nIndex := 0;
IF ipListOfMoversToCheck <> 0 THEN
	THIS^.ipListOfMoversToCheck.ResetIterator();
	WHILE THIS^.ipListOfMoversToCheck.HasNextObject() DO
		
		//Cheack all Movers fill the actposition in the array
		IF ToXpMover(THIS^.ipListOfMoversToCheck.GetNextObject(),ipMover) THEN
			aMoversInterfaceLastCycle[nIndex] 	:= ipMover;
			aMoversPositionLastCycle[nIndex] 	:= ipMover.PositionOnTrack;
			aMoversTrackLastCycle[nIndex]		:= ipMover.CurrentTrack;
			nIndex := nIndex +1;
		END_IF
		
	END_WHILE	
	THIS^.ipListOfMoversToCheck.RestoreIterator();
END_IF
END_METHOD

END_FUNCTION_BLOCK

// COMPONENTs/Optional/Trigger/I_XP_Trigger
INTERFACE I_XP_Trigger  EXTENDS __SYSTEM.IQueryInterface

{attribute 'monitoring':='call'}
PROPERTY AccocietedTrack : I_XP_Track
GET
END_GET
SET
END_SET
END_PROPERTY

{attribute 'monitoring':='call'}
PROPERTY HR : HRESULT
GET
END_GET
END_PROPERTY

PROPERTY ListOfMoversToCheck : I_CH_List
SET
END_SET
END_PROPERTY

{attribute 'monitoring':='call'}
PROPERTY MoverAtTrigger : I_XP_Mover
GET
END_GET
END_PROPERTY

{attribute 'monitoring':='call'}
PROPERTY MoverDetected : BOOL
GET
END_GET
END_PROPERTY

{attribute 'monitoring':='call'}
PROPERTY PositionOnTrack : LREAL
GET
END_GET
SET
END_SET
END_PROPERTY

{attribute 'monitoring':='call'}
PROPERTY TimeStamp : T_DCTIME64;
GET
END_GET
END_PROPERTY

{attribute 'monitoring':='call'}
PROPERTY TriggerDirection : Tc3_Mc3Definitions.MC_Direction
GET
END_GET
SET
END_SET
END_PROPERTY

END_INTERFACE

// COMPONENTs/Optional/Zone/FB_XP_SoretedListOfMover
{attribute 'no_explicit_call' := 'Do not call the body - Stick to OOP'}
// Check zone start to end in positive direktion.
FUNCTION_BLOCK FB_XP_SoretedListOfMover EXTENDS FB_CH_Object IMPLEMENTS I_XP_Zone
VAR
	{attribute 'hide'}
	bInitDone : BOOL;
	{attribute 'hide'}
	ipXpStation : I_XP_Station; //Interface to XPlanar station 
	{attribute 'hide'}
	ipListOfMoversToCheck : CHALET_BaseComponents.I_CH_LIST;
	{attribute 'hide'}
	aMoversInZone : ARRAY [0..(CHALET_BaseComponents.BaseParameterlist.MAX_OBJECTS-1)] OF I_XP_Mover_PLC;
END_VAR

{attribute 'monitoring':='call'}
PROPERTY CtsMoversInZone : UINT
GET
VAR
	nIndex : UDINT;
END_VAR
THIS^.Prepare();//Prepare Time-critical information

//Check array for entrys, exit if fisrt empty arrayindex is found.
FOR nIndex := 0 TO (CHALET_BaseComponents.BaseParameterlist.MAX_OBJECTS-1) DO
	IF (aMoversInZone[nIndex] <> 0) THEN
		CtsMoversInZone := CtsMoversInZone +1;
	ELSE
		RETURN;
	END_IF
END_FOR
END_GET
END_PROPERTY

METHOD FB_init : BOOL
VAR_INPUT
	bInitRetains : BOOL; // if TRUE, the retain variables are initialized (warm start / cold start)
	bInCopyCode : BOOL;  // if TRUE, the instance afterwards gets moved into the copy code (online change)
	
	ipXpStation : I_XP_Station; //Interface to XPlanar station 
	ipListOfMoversToCheck : CHALET_BaseComponents.I_CH_LIST;
END_VAR
VAR_INST
	{attribute 'hide'}
	bFBInitCalledOnce : BOOL; //Do the following code once during start up and not during onlinechange
END_VAR
//Do the following code once during start up and not during onlinechange
IF NOT bFBInitCalledOnce THEN 
	;
END_IF

THIS^.ipXpStation := ipXpStation;
THIS^.ipListOfMoversToCheck := ipListOfMoversToCheck;


bFBInitCalledOnce := TRUE;
END_METHOD

METHOD Initialize : HRESULT
IF THIS^.ipXpStation = 0 THEN
	//No valide interface
	Initialize := E_FAIL;
	RETURN;
END_IF

IF THIS^.ipListOfMoversToCheck = 0 THEN
	//No valide interface
	Initialize := E_FAIL;
	RETURN;
END_IF


bInitDone := TRUE;
Initialize := S_OK;
END_METHOD

{attribute 'monitoring':='call'}
// Return a sorted list of movers in this zone. Index 0 is the mover in Front.
PROPERTY MoversInZone : REFERENCE TO ARRAY [0..(CHALET_BaseComponents.BaseParameterlist.MAX_OBJECTS-1)] OF I_XP_Mover_PLC
GET
THIS^.Prepare();//Prepare Time-critical information

MoversInZone REF= THIS^.aMoversInZone;
END_GET
END_PROPERTY

(* Time-critical information is processed here, which can then be polled via the property every cycle. 
The update method is usually at the end of the program and then it is already 'outdated'. *)
METHOD PRIVATE Prepare : HRESULT
VAR
	nLoopIndex : UDINT;
	ipMoverPlc : I_XP_Mover_PLC;
	ipMover : I_XP_Mover;
	ipPath : I_XP_Path;
	fDistToStart : LREAL;
	aDisanceToStart : ARRAY [0..(CHALET_BaseComponents.BaseParameterlist.MAX_OBJECTS-1)] OF LREAL;
END_VAR
VAR_INST
	{attribute 'hide'}
	nLastUpdatedCycleCount : UDINT;
END_VAR
IF NOT bInitDone OR ipXpStation.AccocietedTrack = 0 THEN
	Prepare := E_FAIL;
	RETURN;
END_IF

//Check if this Cycle the dates are allready prepared
IF nLastUpdatedCycleCount <> TwinCAT_SystemInfoVarList._TaskInfo[THIS^.nTaskIndex].CycleCount THEN
	nLastUpdatedCycleCount := TwinCAT_SystemInfoVarList._TaskInfo[THIS^.nTaskIndex].CycleCount;

	//Clear array
	MEMSET(destAddr:=ADR(aMoversInZone),n:=SIZEOF(aMoversInZone),fillByte:=0);
	
	//Cheack all Movers and generate a sorted list of all mover in this zone.
	THIS^.ipListOfMoversToCheck.ResetIterator();
	WHILE THIS^.ipListOfMoversToCheck.HasNextObject() DO
		//Check each mover in this stations list
		IF __QUERYINTERFACE(THIS^.ipListOfMoversToCheck.GetNextObject(),ipMoverPlc) THEN
			
			//mover and distance are known from this point and are now sorted into the array
			fDistToStart := ipMoverPlc.DistToParentStation;
			ipMoverPlc := ipMoverPlc;
			
			//Check array of movers and decide if the current one is closer to 
			FOR nLoopIndex := 0 TO (CHALET_BaseComponents.BaseParameterlist.MAX_OBJECTS-1) DO
				//empty array position
				IF aMoversInZone[nLoopIndex] = 0 THEN
					aMoversInZone[nLoopIndex] := ipMoverPlc;
					aDisanceToStart[nLoopIndex] := fDistToStart;
					EXIT;
					
				//Closer Mover found, move whole array 	
				ELSIF aDisanceToStart[nLoopIndex] > fDistToStart THEN
					MEMMOVE(srcAddr := ADR(aMoversInZone[nLoopIndex]), destAddr := ADR(aMoversInZone[nLoopIndex+1]), n := (SIZEOF(aMoversInZone[0])*(CHALET_BaseComponents.BaseParameterlist.MAX_OBJECTS-1-nLoopIndex)));
					MEMMOVE(srcAddr := ADR(aDisanceToStart[nLoopIndex]), destAddr := ADR(aDisanceToStart[nLoopIndex+1]), n := (SIZEOF(aDisanceToStart[0])*(CHALET_BaseComponents.BaseParameterlist.MAX_OBJECTS-1-nLoopIndex)));
					aMoversInZone[nLoopIndex] := ipMoverPlc;
					aDisanceToStart[nLoopIndex] := fDistToStart;
					EXIT;
					
				//check next position	
				ELSE 
					;
				END_IF
			END_FOR
		END_IF
	END_WHILE
	THIS^.ipListOfMoversToCheck.RestoreIterator();
END_IF
END_METHOD

METHOD Update : HRESULT
VAR

END_VAR
// Nothing todo in Update. Check Prepare
END_METHOD

END_FUNCTION_BLOCK

// COMPONENTs/Optional/Zone/I_XP_Zone
INTERFACE I_XP_Zone

{attribute 'monitoring':='call'}
PROPERTY CtsMoversInZone : UINT
GET
END_GET
END_PROPERTY

{attribute 'monitoring':='call'}
PROPERTY MoversInZone : REFERENCE TO ARRAY [0..(CHALET_BaseComponents.BaseParameterlist.MAX_OBJECTS-1)] OF I_XP_Mover_PLC // Return a sorted list of movers in this zone. Index 0 is the mover in Front.
GET
END_GET
END_PROPERTY

END_INTERFACE

// COMPONENTs/Optional/I_XP_Path
INTERFACE I_XP_Path  EXTENDS __SYSTEM.IQueryInterface, I_CH_Object

METHOD DistanceToDestiantion : LREAL
VAR_INPUT
	ipTrack : I_XP_Track;
	fPosOnTrack : LREAL;
END_VAR
END_METHOD

{attribute 'monitoring':='call'}
PROPERTY Length : LREAL
GET
END_GET
SET
END_SET
END_PROPERTY

PROPERTY PointerToThis : POINTER TO FB_XP_Path
GET
END_GET
END_PROPERTY

{attribute 'monitoring':='call'}
PROPERTY StationDestination : I_XP_Station
GET
END_GET
SET
END_SET
END_PROPERTY

{attribute 'monitoring':='call'}
PROPERTY StationStart  : I_XP_Station
GET
END_GET
SET
END_SET
END_PROPERTY

{attribute 'monitoring':='call'}
PROPERTY TracksUsed : REFERENCE TO FB_CH_List
GET
END_GET
END_PROPERTY

END_INTERFACE

// COMPONENTs/Optional/FB_XP_Path
{attribute 'enable_dynamic_creation'}
{attribute 'no_explicit_call' := 'Do not call the body - Stick to OOP'}
FUNCTION_BLOCK FB_XP_Path EXTENDS FB_CH_Object IMPLEMENTS I_XP_Path
VAR
	fbTracksUsed : FB_CH_List;
	ipStartStation, ipDestinationStation : I_XP_Station;
	fPathLength : LREAL;
END_VAR

METHOD DistanceToDestiantion : LREAL
VAR_INPUT
	ipTrack : I_XP_Track;
	fPosOnTrack : LREAL;
END_VAR
VAR
	ipTrackTemp : I_XP_Track; 
	bStartTrackFound : BOOL := FALSE;
END_VAR
IF ipTrack = 0 THEN
	//Error -  invalide interface
	DistanceToDestiantion := CHALET_BaseComponents.GVL_Datatypes.cMaxLreal;
	RETURN;
END_IF

IF NOT fbTracksUsed.FindObject(ipTrack) OR fPosOnTrack < 0 OR  fPosOnTrack > ipTrack.Length THEN
	//Error -  position not on track
	DistanceToDestiantion := CHALET_BaseComponents.GVL_Datatypes.cMaxLreal;
	RETURN;
END_IF

//the whole thing works because the tracklist is sorted from start to finish
fbTracksUsed.ResetIterator();
WHILE fbTracksUsed.HasNextObject() DO
	IF ToXpTrack(fbTracksUsed.GetNextObject(),ipTrackTemp) THEN
		//start countion on requestet track
		IF ipTrackTemp = ipTrack OR bStartTrackFound THEN
			bStartTrackFound := TRUE;
			DistanceToDestiantion := DistanceToDestiantion + ipTrackTemp.Length;
 		END_IF
	END_IF
END_WHILE	

DistanceToDestiantion := DistanceToDestiantion - fPosOnTrack;
DistanceToDestiantion := DistanceToDestiantion - THIS^.StationDestination.AccocietedTrack.Length + THIS^.StationDestination.PositionOnTrack;
END_METHOD

{attribute 'monitoring':='call'}
PROPERTY Length : LREAL
GET
Length := THIS^.fPathLength;
END_GET
SET
THIS^.fPathLength := Length;
END_SET
END_PROPERTY

{attribute 'monitoring':='call'}
PROPERTY LUID : STRING //Locally unique identifier
GET
VAR
	sTempName : STRING;
END_VAR
IF ipStartStation <> 0 AND ipDestinationStation <> 0 THEN
	sTempName := CONCAT(sTempName, ipStartStation.LUID);
	sTempName := CONCAT(sTempName, ' to ' );
	sTempName := CONCAT(sTempName, ipDestinationStation.LUID);
	
ELSIF ipStartStation <> 0 THEN
	sTempName := CONCAT(sTempName, ipStartStation.LUID);
	sTempName := CONCAT(sTempName, ' to ?' );

ELSIF ipDestinationStation <> 0 THEN
	sTempName := CONCAT(sTempName, '? to ' );
	sTempName := CONCAT(sTempName, ipDestinationStation.LUID);
	
ELSE 
	sTempName := ' Unknown path';
END_IF


LUID := sTempName;
END_GET
END_PROPERTY

PROPERTY PointerToThis : POINTER TO FB_XP_Path
GET
PointerToThis := ADR(THIS^);
END_GET
END_PROPERTY

{attribute 'monitoring':='call'}
PROPERTY StationDestination : I_XP_Station
GET
StationDestination := THIS^.ipDestinationStation;
END_GET
SET
THIS^.ipDestinationStation := StationDestination;
END_SET
END_PROPERTY

{attribute 'monitoring':='call'}
PROPERTY StationStart  : I_XP_Station
GET
StationStart := THIS^.ipStartStation;
END_GET
SET
THIS^.ipStartStation := StationStart;
END_SET
END_PROPERTY

{attribute 'monitoring':='call'}
PROPERTY TracksUsed : REFERENCE TO FB_CH_List
GET
TracksUsed REF= THIS^.fbTracksUsed;
END_GET
END_PROPERTY

END_FUNCTION_BLOCK

// COMPONENTs/Optional/F_GetDistToPosModulo
FUNCTION F_GetDistToPosModulo : LREAL //This is only working in Positiv Direktion
VAR_INPUT
	fTargedPosition : LREAL;
	fActualPosition : LREAL;
	fModulo 		: LREAL;
END_VAR

VAR

END_VAR

IF fTargedPosition < fActualPosition THEN
	fTargedPosition := fTargedPosition + fModulo;
END_IF

F_GetDistToPosModulo := fTargedPosition - fActualPosition;

END_FUNCTION

// COMPONENTs/Optional/F_InLimitTest
FUNCTION F_InLimitTest : BOOL
VAR_INPUT
	fMinimum 	: LREAL;
	fMaximum 	: LREAL;
	fInput 		: LREAL;
END_VAR

//Normal case
// 9 Max
// 5 Test
// 1 Min
IF fMinimum <= fMaximum THEN
	F_InLimitTest := (fInput >= fMinimum) AND (fInput <= fMaximum);
	
//Modulo case	
// 6 | 6  Max
// 5 | 9  Test
// 8 | 8  Min
ELSIF fMinimum > fMaximum THEN
	F_InLimitTest := NOT((fInput > fMaximum) AND (fInput < fMinimum));
END_IF

END_FUNCTION

// COMPONENTs/Stationen/FB_XP_Station
{attribute 'no_explicit_call' := 'Do not call the body - Stick to OOP'}
(* XPlanar station - n per associated XPlanar. Can be instantiated as an array and/or individually
	The stations are the main component of the application. As soon as the system has been started up and all movers are on the track, the movers are only sent from one station to the next.
	Parameters:
		xPos, yPos 			= Absolute position of the station on the xPlanar.
		ipAccocietedTrack 	= The track on which the station is located. If the XY position is not on this track, the next possible track position is assumed on this track.
		sUniqueName 		= Unique name that may only exist once.
		sTargetGroup 		= A name for a group to which this station belongs. Important for redundant stations
 *)	
FUNCTION_BLOCK FB_XP_Station EXTENDS FB_CH_Object IMPLEMENTS I_XP_Station, I_XP_Station_PLC
VAR
	//optional - To visualize the station position in LiveView
	fbOptionalTrackUsedInLiveView : MC_PlanarTrack;

	{attribute 'hide'}
	bErrorDuringFbInit : BOOL;	//Fatal error - Not possible to reset
	
	{attribute 'hide'}
	bInitDone : BOOL;
	{attribute 'hide'}	
	bTrackIsSetInFbInit : BOOL;
	{attribute 'hide'}	
	bMoversInPlace : BOOL;
	{attribute 'hide'}                   	
	eActiveCommand 		: CHALET_Nc.E_NcAxisCommands := CHALET_Nc.E_NcAxisCommands.None;
	{attribute 'hide'}	
	ipXpSystem : I_XP_System_Registration;
	{attribute 'hide'}
	bReadyToRecvMovers 		: BOOL := TRUE;
	{attribute 'hide'}
	sTargetGroup 				: STRING;
	
	{attribute 'hide'}
	bSuppressDynamicsChange		: BOOL; // Suppress to change the dynamic(Gap+velocity) of passing movers. This is usefull in startup
	{attribute 'hide'}
	fMoverGapAtExit 			: LREAL := XPlanarParameterlist.F_MOVER_MINIMUM_GAP_ON_TRACK; // Every mover that leaves or passes the station gets this new gap as a target.
	{attribute 'hide'}
	fMoverVelocityAtExit		: LREAL; // Every mover that leaves or passes the station gets this new velo as a target.
	
	{attribute 'hide'}	
	fbPositionPlanned : PositionXY; //this is the configured/planned position of the station. set via FB_init. If it is not on the track, the PosOnTrackXY is different
	{attribute 'hide'}	
	fPositionOnTrack : LREAL;
	{attribute 'hide'}
	fbPositionOnTrackXY : PositionXY;	
	{attribute 'hide'}	
	nState_Configuring: INT;
	{attribute 'hide'}	
	ipAccocietedTrack : I_XP_Track;
	{attribute 'hide'}
	nMoverQueueSize 			: UINT;
	{attribute 'hide'}
	fTargetPosWindow			: LREAL := 0.05; //[mm]
	{attribute 'hide'}
	tTargetPosMonitoringTime	: TIME := T#0MS;

	
	(*List of stations*)
	{attribute 'hide'}	
	fbStationsAhead : FB_CH_List;
	{attribute 'hide'}	
	fbStationsBehinde : FB_CH_List;
	
	(*List of paths*)
	{attribute 'hide'}	
	fbListPathAhead : FB_CH_List;
	{attribute 'hide'}
	fbListPathBehind : FB_CH_List;
	
	(* Lists to handle the ownership of movers *)
	{attribute 'hide'}
	fbAssignedMovers 			: FB_CH_List;		// Movers approaching the station. This station is the parent of this movers
	{attribute 'hide'}
	fbFeedback : FB_CH_Feedback;	
	
	//Simulation
	{attribute 'hide'}
	fSimulationProcessDuration 	: LREAL; //[s]
	{attribute 'hide'}
	sSimulationTargedStation	: STRING; //GroupID of the targed station to automatic send after the duration
	
	
	//ipXpSystem Is Not Valid at this point, call the konstruktor again in the FB_Init
	{attribute 'hide'}
	fbTrigger 					: FB_XP_Trigger(ipXpSystem);
	{attribute 'hide'}
	fbSortedListMoversInQueue	: FB_XP_SoretedListOfMover(	ipXpStation := THIS^,
															ipListOfMoversToCheck := fbAssignedMovers );
	{attribute 'hide'}
	fDecisionDistance: LREAL;//[mm]
	
	{attribute 'hide'}
	sFilter : STRING;
END_VAR

METHOD PROTECTED CheckInvalideParameter : HRESULT
VAR
 	ipStation : I_XP_Station;
	fbListOfStationsToCheck : FB_CH_List;
END_VAR
//Get a list of all station whitout this station
fbListOfStationsToCheck.Duplicate(THIS^.ipXpSystem.Stations);
fbListOfStationsToCheck.RemoveObject(THIS^);


fbListOfStationsToCheck.ResetIterator();
WHILE fbListOfStationsToCheck.HasNextObject() DO
	IF ToXpStation(fbListOfStationsToCheck.GetNextObject(), ipStation) THEN
		
		//Check for same positions
		IF (ipStation.PositionOnTrack = THIS^.PositionOnTrack) AND (ipStation.AccocietedTrack = THIS^.AccocietedTrack)  THEN
			//Error two stations have same position on track
			CheckInvalideParameter := E_FAIL;
			RETURN;
		END_IF
		
		//Check same unique id
		IF (ipStation.LUID = THIS^.LUID) THEN
			//Error two stations have same unique id
			CheckInvalideParameter := E_FAIL;
			RETURN;
		END_IF
		
		fbListOfStationsToCheck.RemoveObject(ipStation);
	END_IF
END_WHILE
END_METHOD

METHOD protected GetAccocietedTrack : HRESULT
VAR_INPUT
END_VAR

VAR
	ipTrack : I_XP_Track;
	
	fPosOnTrack, fDist	: LREAL;
	fbPositionXYC : PositionXYC;
	fbPositionXY : PositionXY;
	ipClosestTrack : I_XP_Track;
	fDistClosestTrack : LREAL := CHALET_BaseComponents.GVL_Datatypes.cMaxLreal;
END_VAR
//If track is not defind during FB_init, get closest track 
IF NOT bTrackIsSetInFbInit THEN
	THIS^.ipAccocietedTrack := 0;
	THIS^.ipXpSystem.Tracks.ResetIterator();
	WHILE THIS^.ipXpSystem.Tracks.HasNextObject() DO
		IF ToXpTrack(THIS^.ipXpSystem.Tracks.GetNextObject(),ipTrack) THEN 
			
			fPosOnTrack := ipTrack.PlanarTrack.GetArcLengthClosestTo(geometry:= THIS^.fbPositionPlanned);
			//Get the XYC Pos on track
			ipTrack.PlanarTrack.GetPositionAt(fPosOnTrack, fbPositionXYC);
			//Get radius/ distance to positionTarged
			fbPositionXY.x  := THIS^.fbPositionPlanned.x - fbPositionXYC.x;
			fbPositionXY.y  := THIS^.fbPositionPlanned.y - fbPositionXYC.y;
			fDist := fbPositionXY.GetRadius();
			
			IF fDist < fDistClosestTrack THEN
				fDistClosestTrack := fDist;
				ipClosestTrack := ipTrack;
			END_IF
		END_IF
	END_WHILE
	THIS^.ipXpSystem.Tracks.RestoreIterator();
	
	
	THIS^.ipAccocietedTrack := ipClosestTrack;	
END_IF

// Error - No track found
IF THIS^.ipAccocietedTrack = 0 THEN
	GetAccocietedTrack := E_FAIL;
	RETURN;
END_IF
END_METHOD

METHOD GetDecisionDistance : HRESULT
VAR
	fDistToStartOfTrack : LREAL := CHALET_BaseComponents.GVL_Datatypes.cMaxLreal;
	fDistStationBehind : LREAL := CHALET_BaseComponents.GVL_Datatypes.cMaxLreal;
	
	ipPath : I_XP_Path;
END_VAR
(*
As soon as the mover is closer than this distance, the mover can be sent on to the next one if necessary.
This is the distance from the station to the end of the track or the shortest path to this station. Depending on which is closer. This is to ensure that the mover can no longer be overhauled.
*)
fDistToStartOfTrack := THIS^.PositionOnTrack;

THIS^.PathsBehinde.ResetIterator();
WHILE THIS^.PathsBehinde.HasNextObject() DO
	IF __QUERYINTERFACE(THIS^.PathsBehinde.GetNextObject(), ipPath) THEN
		fDistStationBehind := MIN(fDistStationBehind, ipPath.Length);
	END_IF
END_WHILE
THIS^.PathsBehinde.RestoreIterator();

THIS^.fDecisionDistance := CHALET_BaseComponents.GVL_Datatypes.cMaxLreal;
THIS^.fDecisionDistance := MIN(THIS^.fDecisionDistance, fDistToStartOfTrack);
THIS^.fDecisionDistance := MIN(THIS^.fDecisionDistance, fDistStationBehind);

IF THIS^.fDecisionDistance < 1.0 THEN 
	THIS^.fDecisionDistance := 1.0;
END_IF

GetDecisionDistance := S_OK;
END_METHOD

METHOD protected GetPathsAhead : HRESULT
VAR_INPUT
END_VAR

VAR
	fbPathElementsToCheck : FB_CH_List;
	fbListStationsToGetClosest : FB_CH_List;	
	
	
	ipObject 				: I_CH_Object;
	ipStation,ipStation1,ipStation2 	: I_XP_Station;
	ipTrack					: I_XP_Track; 
	ipLastAddedTrack 		: I_XP_Track;
	ipPath 					: I_XP_Path;
	ipPathCurrentLoop  		: I_XP_Path;
	
	
	pFbPath : POINTER TO FB_XP_Path;
	
	fSeachStartPoint : LREAL;
	nIdx : UDINT;
END_VAR
(*
Check whether there is a station further ahead on this track than this one.
If there is no other station on the track, the previous tracks are filled into a list and searched one after the other to see if they have valid stations. 
If the tracks also have no stations, the track before it is added to the list,...
*)

//Clear list, delete dynamic_creation path objects
WHILE NOT fbListPathAhead.IsEmpty DO
	ipObject := fbListPathAhead.GetRandomObject();
	fbListPathAhead.RemoveObject(ipObject);
	
	__QUERYINTERFACE(ipObject, ipPath) ;
	pFbPath := ipPath.PointerToThis;
	__DELETE(pFbPath);
END_WHILE


//new dynamic_creation path objects
pFbPath := __NEW(FB_XP_Path);
//init path
pFbPath^.StationStart := THIS^;
pFbPath^.TracksUsed.ResetIterator();
pFbPath^.TracksUsed.AddObject(THIS^.AccocietedTrack);

//add to list
fbPathElementsToCheck.AddObject(pFbPath^);

//On first pathsearch get an Station who is further ahead than this
fSeachStartPoint := THIS^.PositionOnTrack;



//While list is not empty
WHILE NOT fbPathElementsToCheck.IsEmpty DO
	__QUERYINTERFACE(fbPathElementsToCheck.GetRandomObject(), ipPathCurrentLoop);
	__QUERYINTERFACE(ipPathCurrentLoop.TracksUsed.GetNextObject(),ipLastAddedTrack);
	
	
	//Closed loop
	IF ipLastAddedTrack.ClosedLoop THEN
		//on closed-loop add all stations of this track to list
		fbListStationsToGetClosest.Duplicate(ipLastAddedTrack.StationsOnTrack);
	
		//remove THIS station from list if more than on station is existing
		IF fbListStationsToGetClosest.Size > 1 THEN
			fbListStationsToGetClosest.RemoveObject(THIS^);
		END_IF
	
		
	
	ELSE
		//Not closed loop	
		//Get a List of all stations on track Position > Startpoint
		ipLastAddedTrack.StationsOnTrack.ResetIterator();
		fbListStationsToGetClosest.Clear();
		WHILE ipLastAddedTrack.StationsOnTrack.HasNextObject() DO
			IF ToXpStation(ipLastAddedTrack.StationsOnTrack.GetNextObject(),ipStation) THEN
				//Add all station ahead to list. on closed-loop add all stations of this track to list
				IF ipStation.PositionOnTrack > fSeachStartPoint THEN
					fbListStationsToGetClosest.AddObject(ipStation);
				END_IF
			END_IF
		END_WHILE	
	END_IF
		
	

	
	//Get closest to startpos(0mm)
	WHILE fbListStationsToGetClosest.Size > 1 DO
		fbListStationsToGetClosest.ResetIterator();
		__QUERYINTERFACE(fbListStationsToGetClosest.GetNextObject(),ipStation1);
		__QUERYINTERFACE(fbListStationsToGetClosest.GetNextObject(),ipStation2);
		
		//If station1 is closer to start than station2, remove station2
		IF 		F_GetDistToPosModulo(fTargedPosition := ipStation1.PositionOnTrack, fActualPosition := fSeachStartPoint, fModulo := ipLastAddedTrack.Length) 
			< 	F_GetDistToPosModulo(fTargedPosition := ipStation2.PositionOnTrack, fActualPosition := fSeachStartPoint, fModulo := ipLastAddedTrack.Length) THEN
			fbListStationsToGetClosest.RemoveObject(ipStation2);
		ELSE	
			fbListStationsToGetClosest.RemoveObject(ipStation1);
		END_IF
	END_WHILE
	
	
	IF fbListStationsToGetClosest.Size = 1 THEN
		//Station FOUND
		__QUERYINTERFACE(fbListStationsToGetClosest.GetRandomObject(), ipStation);
		ipPathCurrentLoop.StationDestination := ipStation;
		
		//Calculate Tracklentgh
		ipPathCurrentLoop.TracksUsed.ResetIterator();
		WHILE ipPathCurrentLoop.TracksUsed.HasNextObject() DO
			IF ToXpTrack(ipPathCurrentLoop.TracksUsed.GetNextObject(),ipTrack) THEN
				ipPathCurrentLoop.Length := ipPathCurrentLoop.Length + ipTrack.Length;
			END_IF
		END_WHILE	
		ipPathCurrentLoop.Length := ipPathCurrentLoop.Length - ipPathCurrentLoop.StationStart.PositionOnTrack;
		ipPathCurrentLoop.Length := ipPathCurrentLoop.Length - ipPathCurrentLoop.StationDestination.AccocietedTrack.Length + ipPathCurrentLoop.StationDestination.PositionOnTrack;
		
		fbListPathAhead.AddObject(ipPathCurrentLoop);
		fbPathElementsToCheck.RemoveObject(ipPathCurrentLoop);
	ELSE
		//Station NOT-FOUND, add the subsequent tracks in the list
		ipLastAddedTrack.TracksAhead.ResetIterator();
		WHILE ipLastAddedTrack.TracksAhead.HasNextObject() DO
			ToXpTrack(ipLastAddedTrack.TracksAhead.GetNextObject(), ipTrack);
			//dublicate current path
			pFbPath := __NEW(FB_XP_Path);
			MEMCPY(destAddr := pFbPath, srcAddr := ipPathCurrentLoop.PointerToThis, n := SIZEOF(FB_XP_Path));
			//Add the new track to fresh created path
			pFbPath^.TracksUsed.AddObject(ipTrack);
			//Add to list to check
			fbPathElementsToCheck.AddObject(pFbPath^);
			
		END_WHILE

		
		//delete current path
		fbPathElementsToCheck.RemoveObject(ipPathCurrentLoop);
		pFbPath := ipPathCurrentLoop.PointerToThis;
		__DELETE(pFbPath);
		
	END_IF

	fSeachStartPoint := -0.1;
END_WHILE
END_METHOD

METHOD protected GetPathsBehind : HRESULT
VAR
	ipThisStation : I_XP_Station;
	ipXpStation : I_XP_Station;
	ipPath		: I_XP_Path;
END_VAR
ipThisStation := THIS^;
fbListPathBehind.Clear();

THIS^.fbStationsBehinde.ResetIterator();
WHILE THIS^.fbStationsBehinde.HasNextObject() DO
	IF __QUERYINTERFACE(THIS^.fbStationsBehinde.GetNextObject(),ipXpStation) THEN
		ipXpStation.PathsAhead.ResetIterator();
		WHILE ipXpStation.PathsAhead.HasNextObject() DO
			IF __QUERYINTERFACE(ipXpStation.PathsAhead.GetNextObject(),ipPath) AND_THEN ipPath.StationDestination = ipThisStation THEN
				//add path to this station to list
				fbListPathBehind.AddObject(ipPath);
			END_IF
		END_WHILE	
	END_IF
END_WHILE
END_METHOD

METHOD PROTECTED GetPosOnTrack : HRESULT
VAR
	fbPositionXYC : PositionXYC;
END_VAR
//GetArcLengthClosestTo track
THIS^.fPositionOnTrack := THIS^.ipAccocietedTrack.PlanarTrack.GetArcLengthClosestTo(geometry:= THIS^.fbPositionPlanned);

//Get the XYC Pos on track
THIS^.ipAccocietedTrack.PlanarTrack.GetPositionAt(THIS^.PositionOnTrack, fbPositionXYC);

//XYC -> XY
THIS^.fbPositionOnTrackXY.SetValuesXY(fbPositionXYC.x,fbPositionXYC.y);


//Check for NaN
IF NOT(THIS^.fPositionOnTrack = THIS^.fPositionOnTrack) THEN
	GetPosOnTrack := E_FAIL;
	RETURN;
END_IF
END_METHOD

METHOD PROTECTED GetStationAhead : HRESULT
VAR
	ipPath 		: I_XP_Path;
END_VAR
fbStationsAhead.Clear();


fbListPathAhead.ResetIterator();
WHILE fbListPathAhead.HasNextObject() DO
	IF __QUERYINTERFACE(fbListPathAhead.GetNextObject(),ipPath) THEN
		//add StationDestination to list
		fbStationsAhead.AddObject(ipPath.StationDestination);
	END_IF
END_WHILE
END_METHOD

METHOD PROTECTED GetStationBehinde : HRESULT
VAR_INPUT
END_VAR
VAR
	ipThisStation : I_XP_Station;
	ipXpStation : I_XP_Station;
	ipXpStationAhead : I_XP_Station;
END_VAR
ipThisStation := THIS^;
fbStationsBehinde.Clear();

//Check each Station
THIS^.ipXpSystem.Stations.ResetIterator();
WHILE THIS^.ipXpSystem.Stations.HasNextObject() DO
	IF __QUERYINTERFACE(THIS^.ipXpSystem.Stations.GetNextObject(),ipXpStation) THEN
		//check the list of stations ahead if this station one is existing
		ipXpStation.StationsAhead.ResetIterator();
		WHILE ipXpStation.StationsAhead.HasNextObject() DO
			IF __QUERYINTERFACE(ipXpStation.StationsAhead.GetNextObject(),ipXpStationAhead) AND_THEN (ipXpStationAhead = ipThisStation) THEN
				//add station to list
				fbStationsBehinde.AddObject(ipXpStation);
			END_IF
		END_WHILE	
	END_IF
END_WHILE	
THIS^.ipXpSystem.Stations.RestoreIterator();
END_METHOD

METHOD SetTrackObjName : HRESULT
VAR
	pObject : ITComObject;
	sName : STRING;
END_VAR
FW_ObjMgr_GetObjectInstance(oid:= THIS^.fbOptionalTrackUsedInLiveView.MCTOPLC_STD.TrackOID, iid:= TC_GLOBAL_IID_LIST.IID_ITComObject, pipUnk:= ADR(pObject));
IF pObject <> 0 THEN
	sName := THIS^.LUID;
	pObject.TcSetObjectName(ADR(sName));
END_IF
END_METHOD

//Call this Methode whith seq 0->99, and wait each step until S_OK is returned
METHOD Configure : HRESULT
VAR_INPUT
	nSeq : UINT; //0->100
END_VAR

VAR_INST
	{attribute 'hide'}
	fbFeedback : MC_PlanarFeedback;	
END_VAR
VAR
	bOptionalTrackUsedInLiveViewIsMapped : BOOL;
	fbPositionXYC : PositionXYC;
END_VAR
bOptionalTrackUsedInLiveViewIsMapped := fbOptionalTrackUsedInLiveView.MCTOPLC_STD.TrackOID <> 0;

CASE nSeq OF
	5:	//Get interface of trackobject
		Configure := THIS^.GetAccocietedTrack();	

	10: //Get closest XY-Position on track
		Configure := THIS^.GetPosOnTrack();
		
	11: //Check id is unique and not multiple stations at same position
		Configure := THIS^.CheckInvalideParameter();		
		
		
	13:	//Init Tigger
		fbTrigger.AccocietedTrack := THIS^.AccocietedTrack;
		fbTrigger.PositionOnTrack := THIS^.PositionOnTrack;
		fbTrigger.ListOfMoversToCheck := THIS^.ipXpSystem.Movers;//All mover
		fbTrigger.TriggerDirection := Tc3_Mc3Definitions. MC_DIRECTION.mcDirectionPositive;
		Configure := fbTrigger.Initialize();
	
	14:	//Init Zone		
		Configure := fbSortedListMoversInQueue.Initialize();	
	
	20: //Fill the list of all paths before this station
		Configure := THIS^.GetPathsAhead();		
		
	25: //Fill the list of all stations before this station
		Configure := THIS^.GetStationAhead();

	30: //Fill the list of all paths behinde this station
		Configure := THIS^.GetStationBehinde();	
			
	35: //Fill the list of all stations behinde this station
		Configure := THIS^.GetPathsBehind();

	40: //Determine the distance from which the station can give a new command to a mover
		Configure := THIS^.GetDecisionDistance();
		

//----------------------------------------------------------------		
//The station can optionally be linked to a track object. this track is then displayed in the live view.
//It takes several cycles to prepare the object
	80: IF bOptionalTrackUsedInLiveViewIsMapped THEN
			fbOptionalTrackUsedInLiveView.Clear(fbFeedback);
		END_IF
		
	81:	//Wait for clearing
		IF bOptionalTrackUsedInLiveViewIsMapped THEN
			IF fbFeedback.Done THEN
				Configure := S_OK;
			ELSIF fbFeedback.Busy THEN
				Configure := S_PENDING;
			ELSIF fbFeedback.Error THEN
				Configure := E_FAIL;
			END_IF	
		END_IF

	82: //Set position 
		IF bOptionalTrackUsedInLiveViewIsMapped THEN
			fbPositionXYC.SetValuesXY(THIS^.PositionOnTrackXY.x, THIS^.PositionOnTrackXY.y);
			fbOptionalTrackUsedInLiveView.AppendPosition(position := fbPositionXYC, commandFeedback:= fbFeedback);	
		END_IF	
	
	83:	//Wait for set position
		IF bOptionalTrackUsedInLiveViewIsMapped THEN
			IF fbFeedback.Done THEN
				Configure := S_OK;
			ELSIF fbFeedback.Busy THEN
				Configure := S_PENDING;
			ELSIF fbFeedback.Error THEN
				Configure := E_FAIL;
			END_IF	
		END_IF
		
	84:	//Set name of "track" to stationsname 
		IF bOptionalTrackUsedInLiveViewIsMapped THEN
 			Configure := SetTrackObjName();
		END_IF
//----------------------------------------------------------------

		
		

	100..CHALET_BaseComponents.GVL_Datatypes.cMaxUint: 
		// 100..MaxUint -> Invalide input
		Configure := E_FAIL;
		
	ELSE 
		//If an step is not defind/used return ok
		Configure := S_OK;
END_CASE


fbOptionalTrackUsedInLiveView.Update();
fbFeedback.Update();
END_METHOD

{attribute 'monitoring':='call'}
PROPERTY CtsEmptySpaceInQueue : UDINT
GET
//Handle UINT Overflow
IF THIS^.fbAssignedMovers.Size >= THIS^.nMoverQueueSize THEN
	CtsEmptySpaceInQueue := 0;
ELSE 
	CtsEmptySpaceInQueue := THIS^.nMoverQueueSize - THIS^.fbAssignedMovers.Size;
END_IF
END_GET
END_PROPERTY

{attribute 'monitoring':='call'}
PROPERTY CtsMoversInQueue : UDINT
GET
CtsMoversInQueue := THIS^.fbAssignedMovers.Size;
END_GET
END_PROPERTY

{attribute 'monitoring':='call'}
PROPERTY MoverQueueSize : UINT
GET
MoverQueueSize := THIS^.nMoverQueueSize;
END_GET
SET
THIS^.nMoverQueueSize := MoverQueueSize;
END_SET
END_PROPERTY

{attribute 'monitoring':='call'}
PROPERTY MoversInPlace : BOOL
GET
THIS^.Prepare();//Prepare time-critical information, if not already done


MoversInPlace := bMoversInPlace;
END_GET
END_PROPERTY

{attribute 'monitoring':='call'}
// Return a sorted list of movers in this zone. Index 0 is the mover in Front
PROPERTY MoversInQueue : REFERENCE TO ARRAY [0..(CHALET_BaseComponents.BaseParameterlist.MAX_OBJECTS-1)] OF I_XP_Mover_PLC
GET
MoversInQueue REF= THIS^.fbSortedListMoversInQueue.MoversInZone;
END_GET
END_PROPERTY

{attribute 'monitoring':='call'}
//prevent further movers from entering the station, 
//e.g. to prevent a collision. All movers that are already moving to reach this station will be stopped with a stop 
//and restarted with Ready True.
PROPERTY ReadyToRecvMovers : BOOL
GET
ReadyToRecvMovers := bReadyToRecvMovers;
END_GET
SET
VAR
	ipEachMover : I_XP_Mover;
END_VAR
//Change to Not Ready:
IF (ReadyToRecvMovers = FALSE) AND (bReadyToRecvMovers <> ReadyToRecvMovers) THEN
	//halt all movers on the way
	fbAssignedMovers.ResetIterator();
	WHILE fbAssignedMovers.HasNextObject() DO
		IF ToXpMover(fbAssignedMovers.GetNextObject(),ipEachMover) THEN
			ipEachMover.Halt();	
		END_IF	
	END_WHILE
END_IF

//Change to Ready:
IF (ReadyToRecvMovers = TRUE) AND (bReadyToRecvMovers <> ReadyToRecvMovers) THEN
	//all movers that are on the way have probably been stopped before. when reactivated, the last move command is sent again.
	fbAssignedMovers.ResetIterator();
	WHILE fbAssignedMovers.HasNextObject() DO
		IF ToXpMover(fbAssignedMovers.GetNextObject(),ipEachMover) THEN
			ipEachMover.MoveOnTrack(ipTrack 	:= ipEachMover.LastCmdTargedTrack ,
									fPosition	:= ipEachMover.LastCmdTargedPosition,
									fGap		:= ipEachMover.LastCmdTargedGap);
		END_IF	
	END_WHILE
END_IF

//Store new status
bReadyToRecvMovers := ReadyToRecvMovers;
END_SET
END_PROPERTY

METHOD SendMoversToStation : I_CH_Feedback //All movers in the station are sent to this destination
VAR_INPUT
	sTargetStation: STRING;//unique station name or group of stations
END_VAR
VAR
	nIdx : UDINT;
	ipXpMover : I_XP_Mover;
END_VAR
IF THIS^.fbFeedback.Error THEN
	//Error active/not ready
	THIS^.fbFeedback.LastCommandAccepted	:= FALSE;
	RETURN;
END_IF

//Invalide targed
IF sTargetStation = '' THEN
	THIS^.fbFeedback.LastCommandAccepted	:= FALSE;
	RETURN;
END_IF

//Movers have not reached station and can not send away until complet
IF NOT THIS^.MoversInPlace THEN
	THIS^.fbFeedback.LastCommandAccepted	:= FALSE;
	RETURN;
END_IF

//Send all Queued movers away by changing the targed station destination
FOR nIdx := 0 TO nMoverQueueSize-1 DO
	IF THIS^.MoversInQueue[nIdx] <> 0 AND_THEN __QUERYINTERFACE(THIS^.MoversInQueue[nIdx],ipXpMover) THEN
		ipXpMover.TargetStation := sTargetStation;		
	END_IF
	
	THIS^.fbFeedback.LastCommandAccepted	:= TRUE;;
END_FOR

SendMoversToStation := THIS^.fbFeedback;
END_METHOD

{attribute 'monitoring':='call'}
//Suppress to change the dynamic(Gap+velocity) of passing movers. This is usefull in startup
PROPERTY SuppressDynamicsChange : BOOL
GET
SuppressDynamicsChange := bSuppressDynamicsChange;
END_GET
SET
bSuppressDynamicsChange := SuppressDynamicsChange;
END_SET
END_PROPERTY

{attribute 'monitoring':='call'}
PROPERTY TargetGroupe : STRING
GET
TargetGroupe := THIS^.sTargetGroup;
END_GET
END_PROPERTY

{attribute 'monitoring':='call'}
//A time that is waited as soon as the mover is in the station (including the monitoring window) before “MoversInPlace” is set. e.g. used to stabilize the workpiece
PROPERTY TargetPosMonitoringTime : TIME
GET
TargetPosMonitoringTime := tTargetPosMonitoringTime;
END_GET
SET
tTargetPosMonitoringTime := TargetPosMonitoringTime;
END_SET
END_PROPERTY

{attribute 'monitoring':='call'}
//How many mm before the mover reaches the position is “MoversInPlace” set for the process. 
//This distance can also be set very large (e.g. 100mm) for moving past without stopping.
PROPERTY TargetPosWindow : LREAL
GET
TargetPosWindow := fTargetPosWindow;
END_GET
SET
fTargetPosWindow := TargetPosWindow;
END_SET
END_PROPERTY

{attribute 'monitoring':='call'}
PROPERTY ProcessSimulationActive : BOOL
GET
ProcessSimulationActive := THIS^.fSimulationProcessDuration > 0;
END_GET
END_PROPERTY

METHOD PROTECTED Simulation : HRESULT
VAR_INST
	tonSimulationDelay : TON;
END_VAR
//Automatic send mover to next station in Simulation
//If a valid time (>0seconds) is set and the configured destination station exists, then the movers will be sent away automatically after this time from now on.
tonSimulationDelay.IN 	:= THIS^.ipXpSystem.Enabled AND THIS^.MoversInPlace AND THIS^.ProcessSimulationActive;
tonSimulationDelay.PT	:= LREAL_TO_TIME(THIS^.fSimulationProcessDuration*1000.0);
tonSimulationDelay();
IF tonSimulationDelay.Q THEN
	THIS^.SendMoversToStation(sTargetStation := THIS^.sSimulationTargedStation);
END_IF
END_METHOD

//If a valid time (>0seconds) is set and the configured destination station exists, then the movers will be sent away automatically after this time from now on.
METHOD SimulationMode : HRESULT
VAR_INPUT
	fProcessDuration 		: LREAL; //[s]
	sTargedStation	: STRING; //Group of the targed station to automatic send after the duration
END_VAR
VAR
	ipStation	: I_CH_Object;
	ipXpSystemPlc : I_XP_System_PLC;
	bValideStation : BOOL;
END_VAR
bValideStation := __QUERYINTERFACE(THIS^.ipXpSystem,ipXpSystemPlc) AND ipXpSystemPlc <> 0 AND_THEN ipXpSystemPlc.CheckTargetExists(sTargedStation);

IF (fProcessDuration > 0) AND bValideStation THEN
	//Valide config
	THIS^.fSimulationProcessDuration 	:=	fProcessDuration;
	THIS^.sSimulationTargedStation 		:=	sTargedStation;
	SimulationMode := S_OK;
ELSE
	//Simulation disabled
	THIS^.fSimulationProcessDuration 	:=	0;
	THIS^.sSimulationTargedStation 		:=	'';
	SimulationMode := S_FALSE;
END_IF
END_METHOD

{attribute 'monitoring':='call'}
//Track on which the station is located
PROPERTY AccocietedTrack : I_XP_Track
GET
AccocietedTrack := THIS^.ipAccocietedTrack;
END_GET
END_PROPERTY

METHOD AddMoverToQueue : HRESULT
VAR_INPUT
	ipMover : I_XP_Mover;
END_VAR
VAR
	ipObject : I_CH_Object;
END_VAR
//Get I_CH_Objekt of mover to put it in to a list.
IF ipMover <> 0 AND_THEN __QUERYINTERFACE(ipMover,ipObject) THEN
	//Add in List of Movers in this station
	THIS^.fbAssignedMovers.AddObject(ipObject);
	
	//Handover information in Mover
	ipMover.ParentStation := (THIS^);

	AddMoverToQueue := S_OK;
ELSE
	AddMoverToQueue := E_FAIL;;	
END_IF
END_METHOD

{attribute 'monitoring':='call'}
//List of movers managed by this station
PROPERTY AssignedMovers : I_CH_List
GET
AssignedMovers := THIS^.fbAssignedMovers;
END_GET
END_PROPERTY

METHOD DeleteMoversQueue : HRESULT
VAR
	ipTempMover : I_XP_Mover;
END_VAR
//Delete intormation in linked mover
THIS^.fbAssignedMovers.ResetIterator();
WHILE THIS^.fbAssignedMovers.HasNextObject() DO
	IF ToXPMover(THIS^.fbAssignedMovers.GetNextObject(),ipTempMover) THEN
		ipTempMover.ParentStation := 0;
	END_IF	
END_WHILE

//Clear list
fbAssignedMovers.Clear();

DeleteMoversQueue := S_OK;
END_METHOD

METHOD FB_exit : BOOL
VAR_INPUT
	bInCopyCode : BOOL; // if TRUE, the exit method is called for exiting an instance that is copied afterwards (online change).
END_VAR
VAR
	pFbPath : POINTER TO FB_XP_Path;
	ipObject : I_CH_Object;
	ipPath : I_XP_Path;
END_VAR
//Clear list, delete dynamic_creation path objects
WHILE NOT THIS^.fbListPathAhead.IsEmpty DO
	ipObject := fbListPathAhead.GetRandomObject();
	fbListPathAhead.RemoveObject(ipObject);
	
	__QUERYINTERFACE(ipObject, ipPath) ;
	pFbPath := ipPath.PointerToThis;
	__DELETE(pFbPath);
END_WHILE
END_METHOD

METHOD FB_init : BOOL
VAR_INPUT
	bInitRetains : BOOL; // if TRUE, the retain variables are initialized (warm start / cold start)
	bInCopyCode : BOOL;  // if TRUE, the instance afterwards gets moved into the copy code (online change)
	
	ipSystem 			: I_CH_Object;
	ipAccocietedTrack 	: I_XP_Track;//track on which the station is located
	sUniqueName			: STRING;		//expl.:'Loading' unique identification for this station
	sTargetGroup		: STRING;	//to which group of stations does this station belong? e.g. several stations can belong to one 'Infeed' if this is implemented redundantly.
	nMoverQueueSize 	: UINT;
	xPos, yPos			: LREAL; 	
END_VAR

VAR_INST
	{attribute 'hide'}
	bFBInitCalledOnce : BOOL; //Do the following code once during start up and not during onlinechange
END_VAR

VAR 



END_VAR
//Do the following code once during start up and not during onlinechange
IF NOT bFBInitCalledOnce THEN 
	
	(* Register to the Xplanar System
	   1. Test if the interface exists
	   2. Test if the object implements a "System for Mover" interface 
	*)
	IF ipSystem <> 0 AND_THEN __QUERYINTERFACE(ipSystem,THIS^.ipXpSystem) THEN
		THIS^.ipXpSystem.RegisterStation(THIS^);
	ELSE
		bErrorDuringFbInit := TRUE;
	END_IF

	
	// 0 = get closest track (in step configure)
	IF ipAccocietedTrack <> 0 THEN
		THIS^.ipAccocietedTrack := ipAccocietedTrack;
		bTrackIsSetInFbInit := TRUE;
	END_IF
	 
	
	//"" is maybe entered in an waiting or dynamic station and the name is not important
	IF sUniqueName <> '' THEN 
		THIS^.fbSourceInfo.sName := sUniqueName;
	ELSE
		sUniqueName := THIS^.fbSourceInfo.sName;
	END_IF

	
	//"" is maybe entered in an waiting or dynamic station and the name is not important
	IF sTargetGroup <> '' THEN 
		THIS^.sTargetGroup := sTargetGroup;
	ELSE
		THIS^.sTargetGroup := THIS^.fbSourceInfo.sName;
	END_IF

	
	THIS^.nMoverQueueSize 		:= nMoverQueueSize;
	THIS^.fbPositionPlanned.x 	:= xPos;
	THIS^.fbPositionPlanned.y 	:= yPos;


	THIS^.fbTrigger.FB_init(FALSE,FALSE, THIS^.ipXpSystem);

END_IF

bFBInitCalledOnce := TRUE;
END_METHOD

{attribute 'monitoring':='call'}
PROPERTY Feedback : I_CH_Feedback
GET
Feedback := THIS^.fbFeedback;
END_GET
END_PROPERTY

{attribute 'monitoring':='call'}
//Filter content, movers with one of these targets may not approach or drive over the station
PROPERTY Filter : STRING
GET
Filter := sFilter;
END_GET
SET
sFilter := Filter;
END_SET
END_PROPERTY

METHOD Initialize : HRESULT
VAR
	ipEachStationAhead : I_XP_Station;
END_VAR
VAR_INST
	//This error cannot be reset. Requires a reset cold
	{attribute 'hide'}	
	fbInitError : FB_TcAlarm;
	{attribute 'hide'}	
	fbMissingInterfaceAlarm : FB_TcAlarm;
END_VAR
//Check Error during FB_Init
IF THIS^.bErrorDuringFbInit THEN
	IF NOT fbInitError.bRaised THEN 
		//This error cannot be reset. Requires a reset cold
		fbInitError.CreateEx(stEventEntry:=TC_EVENTS.CHALET_XTS_Events.ErrorFBinit, ipSourceInfo := THIS^.fbSourceInfo, bWithConfirmation := FALSE);
		fbInitError.Raise(0);
	END_IF
	Initialize:= E_FAIL;
	THIS^.fbFeedback.HR := Initialize;
	RETURN;
END_IF	

//Interface to System is missing
IF THIS^.ipXpSystem = 0 THEN
	IF NOT fbMissingInterfaceAlarm.bRaised THEN 
		//This error cannot be reset. Requires a reset cold
		fbMissingInterfaceAlarm.CreateEx(stEventEntry:=TC_EVENTS.CHALET_XTS_Events.InitializationInvalideParameter, ipSourceInfo := THIS^.fbSourceInfo, bWithConfirmation := FALSE);
		fbMissingInterfaceAlarm.Raise(0);
	END_IF
	Initialize := E_FAIL;
	THIS^.fbFeedback.HR := Initialize;
	RETURN;
END_IF


IF NOT THIS^.bInitDone THEN
	//Busy
	Initialize:= S_PENDING;
	
	//Clean up
	THIS^.DeleteMoversQueue();


	bInitDone := TRUE;
ELSE
	//Done
	Initialize:= S_OK;
END_IF


THIS^.fbFeedback.ActiveCommand 		:= TO_STRING(CHALET_NC.E_NcAxisCommands.Initialize);
THIS^.eActiveCommand 				:= CHALET_NC.E_NcAxisCommands.Initialize;
THIS^.fbFeedback.LastCommandAccepted:= TRUE;	
//Set done or keep in busy state	
THIS^.fbFeedback.HR := Initialize;
END_METHOD

{attribute 'monitoring':='call'}
//[mm] Every mover that leaves or passes the station gets this new gap as a target.
PROPERTY MoverGapAtExit : LREAL
GET
MoverGapAtExit := fMoverGapAtExit;
END_GET
SET
IF MoverGapAtExit < XPlanarParameterlist.F_MOVER_MINIMUM_GAP_ON_TRACK THEN
	MoverGapAtExit := XPlanarParameterlist.F_MOVER_MINIMUM_GAP_ON_TRACK;
END_IF

fMoverGapAtExit := MoverGapAtExit;
END_SET
END_PROPERTY

{attribute 'monitoring':='call'}
 //[mm/s] Every mover that leaves or passes the station gets this new velocity as a target.
PROPERTY MoverVelocityAtExit : LREAL
GET
MoverVelocityAtExit := fMoverVelocityAtExit;
END_GET
SET
fMoverVelocityAtExit := MoverVelocityAtExit;
END_SET
END_PROPERTY

PROPERTY OID : OTCID
GET
OID := THIS^.fbOptionalTrackUsedInLiveView.MCTOPLC_STD.TrackOID;
END_GET
END_PROPERTY

{attribute 'monitoring':='call'}
//List of paths that lead to stations before this station
PROPERTY PathsAhead : I_CH_List
GET
PathsAhead := THIS^.fbListPathAhead;
END_GET
END_PROPERTY

{attribute 'monitoring':='call'}
//List of paths that lead to stations behind this station
PROPERTY PathsBehinde : I_CH_List
GET
PathsBehinde := THIS^.fbListPathBehind;
END_GET
END_PROPERTY

{attribute 'monitoring':='call'}
//[mm] from the beginning of the assigned track
PROPERTY PositionOnTrack : LREAL
GET
PositionOnTrack := THIS^.fPositionOnTrack;
END_GET
END_PROPERTY

{attribute 'monitoring':='call'}
//Position on the assigned track
PROPERTY PositionOnTrackXY : REFERENCE TO PositionXY
GET
PositionOnTrackXY REF= THIS^.fbPositionOnTrackXY;
END_GET
END_PROPERTY

{attribute 'monitoring':='call'}
//Planned position, not necessarily on the track
PROPERTY PositionXY : REFERENCE TO  PositionXY
GET
PositionXY REF= THIS^.fbPositionPlanned;
END_GET
END_PROPERTY

(* 
	Use this Methode to calculate time sensitive date once each cycle. Example: read analog input and convert before do get Signal propertie
*)
METHOD PROTECTED Prepare : HRESULT
VAR_INST
	{attribute 'hide'}	
	nLastUpdatedCycleCount : UDINT;
END_VAR

VAR
	nLoopIndex : UINT;
	fExpectedDistanceToParent : LREAL;
	nCycleTime_ms : UDINT;
	bMoverInQueue : BOOL;
	bTempMoverInPosition : BOOL;
	bTempMoverVeloZero : BOOL;
	bTempMoverInMonitoringTime : BOOL;
	bTempMoverThisStationAsTarged : BOOL;
END_VAR
VAR_INST
	{attribute 'hide'}
	nCycleCountInPos : UDINT;
END_VAR
//Check if this Cycle the dates are allready prepared. This is important for time sensitive informations.
IF nLastUpdatedCycleCount <> TwinCAT_SystemInfoVarList._TaskInfo[THIS^.TaskIndex].CycleCount THEN
	nLastUpdatedCycleCount := TwinCAT_SystemInfoVarList._TaskInfo[THIS^.TaskIndex].CycleCount ;


	(* Check if mover is in place. Time and Position window *)
	//If queuesize is zero, mover is never in place.
	IF nMoverQueueSize = 0 OR THIS^.ipAccocietedTrack = 0 OR NOT ipXpSystem.Enabled THEN
		THIS^.bMoversInPlace := FALSE;
		nCycleCountInPos := 0;
	ELSE
		//Get this task cycle Count and time 
		nCycleTime_ms := TwinCAT_SystemInfoVarList._TaskInfo[THIS^.nTaskIndex].CycleTime(*100ns*) / 10_000 ;
		
		bTempMoverInPosition := TRUE; bTempMoverVeloZero := TRUE; bTempMoverThisStationAsTarged := TRUE;
		fExpectedDistanceToParent := 0;
		FOR nLoopIndex := 0 TO (THIS^.nMoverQueueSize-1) DO
			IF THIS^.fbSortedListMoversInQueue.MoversInZone[nLoopIndex] <> 0 THEN
				//Check position and Gap - 1 mover do not have a gap
				IF nLoopIndex <> 0 THEN
					fExpectedDistanceToParent := fExpectedDistanceToParent + THIS^.fbSortedListMoversInQueue.MoversInZone[nLoopIndex].LastCmdTargedGap;
				END_IF
				bMoverInQueue		:= TRUE;
				bTempMoverInPosition := bTempMoverInPosition AND (ABS(THIS^.fbSortedListMoversInQueue.MoversInZone[nLoopIndex].DistToParentStation - fExpectedDistanceToParent) <= fTargetPosWindow );
				bTempMoverVeloZero := bTempMoverVeloZero AND (THIS^.fbSortedListMoversInQueue.MoversInZone[nLoopIndex].PlanarMover.MCTOPLC.SETONTRACK.SetVelo = 0.0);
				bTempMoverThisStationAsTarged := bTempMoverThisStationAsTarged AND ((THIS^.fbSortedListMoversInQueue.MoversInZone[nLoopIndex].TargetStation = THIS^.TargetGroupe) OR (THIS^.fbSortedListMoversInQueue.MoversInZone[nLoopIndex].TargetStation = THIS^.LUID));
			ELSE
				//Missing mover in queue
				bMoverInQueue := FALSE;
				EXIT;
			END_IF
		END_FOR
			
		//start time if mover position is ok
		IF bTempMoverInPosition  THEN
			nCycleCountInPos := nCycleCountInPos + 1;
		ELSE
			nCycleCountInPos := 0;
		END_IF
		
		bTempMoverInMonitoringTime := (UDINT_TO_TIME(nCycleCountInPos * nCycleTime_ms) >= tTargetPosMonitoringTime);
				
		THIS^.bMoversInPlace := bMoverInQueue AND bTempMoverInPosition AND bTempMoverInMonitoringTime AND bTempMoverThisStationAsTarged;// AND bTempMoverVeloZero;
	END_IF
	
	
	
	
	
	
	
	
END_IF
END_METHOD

METHOD SearchNextBestStationByName : ST_PathFinder_1
VAR_INPUT
	sTargedStation : STRING; //unique station name or group of stations
	nPermittedSearchDepth : UINT;
	bCallFromExternal: BOOL; //set to true for an external call. set to false for a recursive call
END_VAR

VAR_STAT	
	ipWhoIsAsking	: I_XP_Station;
	fbListOfEvaluatedStations : CHALET_BaseComponents.FB_CH_List;
END_VAR

VAR
	nRemainingSearchDepth 			: UINT;
	ipPath							: I_XP_Path;
	ipThisStation 					: I_XP_Station;
	ipDestiantionStation			: I_XP_Station;
	ipStation 						: I_XP_Station;
	stPathTemp, stPathShortest		: ST_PathFinder_1;
	bIamTheAsker					: BOOL;
	bTargetFoundOnThisPath			: BOOL;
	bStationIsOnlyForDynamicChanges : BOOL;
	bStationIsFull					: BOOL;
	bStationHanMoreMoverThanAllowed : BOOL;
	bStationHasAFreePlaceInQueue 	: BOOL;
	bStationIsNotReadyToRecvMovers	: BOOL;
	bAnyFreeStationOfThisTarged		: BOOL;
	//bFilterOfStationDoesNotAllowThisMover : BOOL;
	//fShortestPath 					: LREAL := CHALET_BaseComponents.GVL_Datatypes.cMaxLreal;
	fDistShortestButNotReady		: LREAL := CHALET_BaseComponents.GVL_Datatypes.cMaxLreal;
	bRequestedStation : BOOL;
END_VAR
VAR_INST
	//Store the last value if this station gets multiple request from same asking station
	stLastReturnValue : ST_PathFinder_1;
	fbRouteToParent : FB_CH_List;
	bLastResultValide : BOOL;
END_VAR
ipThisStation := (THIS^);

//Invalide input
IF sTargedStation = '' THEN
	//Error
	searchNextBestStationByName.bTargetFound := FALSE;
	searchNextBestStationByName.ipBestStation := 0;
	searchNextBestStationByName.fDistToTarged := 0.0;
	fbRouteToParent.Clear();
	stPathShortest.ipRouteToParent	:= fbRouteToParent;
	RETURN;
END_IF

//Filter of this station does not allow the current station - this is not a valide path. Only if this station is not the asker
IF ((THIS^.Filter <> '') AND (THIS^.Filter <> sTargedStation) AND NOT bCallFromExternal) THEN
	searchNextBestStationByName.bTargetFound := FALSE;
	searchNextBestStationByName.ipBestStation := 0;
	searchNextBestStationByName.fDistToTarged := 0.0;
	fbRouteToParent.Clear();
	stPathShortest.ipRouteToParent	:= fbRouteToParent;
	RETURN;
END_IF

// New search command - Reset list of evaluated stations in first search routine
IF bCallFromExternal THEN
	ipWhoIsAsking := ipThisStation;
	fbListOfEvaluatedStations.Clear();
	
	//Have any of the stations I'm looking a free space in queue somewhere on the track?
	//Otherwise, verify whether my new station is really closer than my current location. -> Prevent the mover from being sent via an alternative track in the loop
	THIS^.ipXpSystem.Stations.ResetIterator();
	WHILE THIS^.ipXpSystem.Stations.HasNextObject() DO
		IF __QUERYINTERFACE(THIS^.ipXpSystem.Stations.GetNextObject(), ipStation) THEN
			bRequestedStation := (ipStation.LUID = sTargedStation)OR(ipStation.TargetGroupe = sTargedStation);
			bAnyFreeStationOfThisTarged := bAnyFreeStationOfThisTarged OR(bRequestedStation AND ipStation.CtsEmptySpaceInQueue > 0 AND ipStation.ReadyToRecvMovers);
		END_IF
	END_WHILE
	THIS^.ipXpSystem.Stations.RestoreIterator();
END_IF

//Has the maximum search depth been reached?
nRemainingSearchDepth := nPermittedSearchDepth - 1;
IF nRemainingSearchDepth = 0 THEN
	searchNextBestStationByName.bTargetFound := FALSE;
	searchNextBestStationByName.ipBestStation := 0;
	searchNextBestStationByName.fDistToTarged := CHALET_BaseComponents.GVL_Datatypes.cMaxLreal;
	stPathShortest.ipRouteToParent	:= fbRouteToParent;
	stLastReturnValue := searchNextBestStationByName;
	RETURN;
END_IF

//Check whether the station has already been scanned
IF fbListOfEvaluatedStations.FindObject(THIS^) THEN
	IF bLastResultValide THEN
		searchNextBestStationByName := stLastReturnValue;
	ELSE
		SearchNextBestStationByName.bTargetFound := FALSE;
	END_IF
	RETURN;
END_IF

//Create a list with every station that has already been checked. 
//Otherwise it can happen with loops and switches that a route is checked several times.
fbListOfEvaluatedStations.AddObject(THIS^);

//Start a new list
fbRouteToParent.Clear();

//Reset last stored path information this is a new request
stLastReturnValue := SearchNextBestStationByName;
bLastResultValide := FALSE;

//Is the station not aware of any other stations in front of it?
IF THIS^.fbStationsAhead.Size = 0 THEN
	searchNextBestStationByName.bTargetFound := FALSE;
	searchNextBestStationByName.ipBestStation := 0;
	searchNextBestStationByName.fDistToTarged := CHALET_BaseComponents.GVL_Datatypes.cMaxLreal;
	stPathShortest.ipRouteToParent	:= fbRouteToParent;
	stLastReturnValue := searchNextBestStationByName;
	bLastResultValide := TRUE;
	RETURN;
END_IF

//Check if the requested station is this one. And not the station who is searching
IF ((THIS^.TargetGroupe = sTargedStation OR THIS^.LUID = sTargedStation) AND (ipWhoIsAsking <> ipThisStation)) THEN
	//FOUND
	stPathShortest.bTargetFound 	:= TRUE;
	stPathShortest.ipBestStation 	:= THIS^;
	stPathShortest.fDistToTarged 	:= 0.0;
	stPathShortest.ipRouteToParent	:= fbRouteToParent;
	fDistShortestButNotReady 		:= 0.0;
ELSE
	//Check the stations ahead if a movement to targed station is posible. Multiple stations incase of an switch.
	THIS^.fbListPathAhead.ResetIterator();
	WHILE THIS^.fbListPathAhead.HasNextObject() DO
		IF __QUERYINTERFACE(THIS^.fbListPathAhead.GetNextObject(),ipPath) AND_THEN ipPath.StationDestination <> 0 THEN
			ipDestiantionStation := ipPath.StationDestination;
			stPathTemp := ipDestiantionStation.searchNextBestStationByName(sTargedStation := sTargedStation, nPermittedSearchDepth := nRemainingSearchDepth, bCallFromExternal := FALSE);	
			stPathTemp.fDistToTarged := stPathTemp.fDistToTarged + ipPath.Length;
			
			//the information that we are on a valid path is set if a path to destination was detected
			bTargetFoundOnThisPath := bTargetFoundOnThisPath OR stPathTemp.bTargetFound;
	
			// Get the shortest way to targed, ignore that maybe not ready
			IF stPathTemp.bTargetFound  AND stPathTemp.fDistToTarged < fDistShortestButNotReady THEN
				fDistShortestButNotReady := stPathTemp.fDistToTarged;				
			END_IF

			//if a path is found with a valid in-between position, get the shortest path
			IF stPathTemp.bTargetFound AND stPathTemp.ipBestStation <> 0 AND stPathTemp.fDistToTarged < stPathShortest.fDistToTarged THEN
				fbRouteToParent.Duplicate(stPathTemp.ipRouteToParent);
				fbRouteToParent.AddObject(ipPath);
				stPathShortest := stPathTemp;
			END_IF
		END_IF
	END_WHILE
	stPathShortest.bTargetFound := bTargetFoundOnThisPath;
	
	//Abort - not a valide path
	IF NOT stPathShortest.bTargetFound THEN
		searchNextBestStationByName.bTargetFound := FALSE;
		searchNextBestStationByName.ipBestStation := 0;
		searchNextBestStationByName.fDistToTarged := CHALET_BaseComponents.GVL_Datatypes.cMaxLreal;
		stLastReturnValue := searchNextBestStationByName;
		bLastResultValide := TRUE;
		RETURN;
	END_IF
END_IF


//evaluate whether the current best station should be overwritten by this one
bIamTheAsker					:= bCallFromExternal;
bStationHanMoreMoverThanAllowed := (THIS^.CtsMoversInQueue > THIS^.nMoverQueueSize); //Maybe during statup if all movers are forced to station x.	
bStationIsFull					:= (THIS^.CtsEmptySpaceInQueue = 0) AND NOT (THIS^.nMoverQueueSize = 0);
bStationHasAFreePlaceInQueue 	:= (THIS^.CtsEmptySpaceInQueue > 0);
bStationIsOnlyForDynamicChanges := (THIS^.nMoverQueueSize = 0);
bStationIsNotReadyToRecvMovers	:= ( NOT THIS^.bReadyToRecvMovers); 

//End of search. Return found station
IF bIamTheAsker THEN
	
	//Special situation no target station in the entire system not ready
	//Have any of the stations I'm looking a free space in queue somewhere on the track?
	//Otherwise, verify whether my new station is really closer than my current location. -> Prevent the mover from being sent via an alternative track in the loop
	IF (NOT bAnyFreeStationOfThisTarged) AND (fDistShortestButNotReady < stPathShortest.fDistToTarged) THEN
		//Stay on this station
		searchNextBestStationByName.bTargetFound := stPathShortest.bTargetFound;
		searchNextBestStationByName.ipBestStation := 0;
		searchNextBestStationByName.fDistToTarged := 0.0;
		searchNextBestStationByName.ipRouteToParent := 0;
	ELSE
		//Return found station
		searchNextBestStationByName.bTargetFound := stPathShortest.bTargetFound;
		searchNextBestStationByName.ipBestStation := stPathShortest.ipBestStation;
		searchNextBestStationByName.fDistToTarged := stPathShortest.fDistToTarged;
		searchNextBestStationByName.ipRouteToParent := fbRouteToParent;
	END_IF


//Is THIS Station a "Dynamic change station" (Queuesize = 0) and has only the purpose tho change the gap of passing movers.
//in this case, the current path should be left as it is. the station is ignored,
ELSIF bStationIsOnlyForDynamicChanges THEN
	searchNextBestStationByName.bTargetFound := stPathShortest.bTargetFound;
	searchNextBestStationByName.ipBestStation := stPathShortest.ipBestStation;
	searchNextBestStationByName.fDistToTarged := stPathShortest.fDistToTarged;
	searchNextBestStationByName.ipRouteToParent := fbRouteToParent;


//This station is full, no movement posible. Do not evaluate if this station is the asker.(Dont care if my own station is full atm.)
ELSIF bStationIsFull OR bStationHanMoreMoverThanAllowed OR bStationIsNotReadyToRecvMovers OR bStationIsOnlyForDynamicChanges THEN
	searchNextBestStationByName.bTargetFound := TRUE;
	searchNextBestStationByName.ipBestStation := 0;
	searchNextBestStationByName.fDistToTarged := fDistShortestButNotReady;
	searchNextBestStationByName.ipRouteToParent := 0;
	
	
//This station in an valide an good targed for the mover. return this station
	ELSE
	searchNextBestStationByName.bTargetFound := TRUE;
	searchNextBestStationByName.ipBestStation := (THIS^);
	searchNextBestStationByName.fDistToTarged := fDistShortestButNotReady;
	searchNextBestStationByName.ipRouteToParent := 0;
END_IF

//Store the last value 
//if this station gets multiple request from same asking station return this
stLastReturnValue := SearchNextBestStationByName;
bLastResultValide := TRUE;
END_METHOD

{attribute 'monitoring':='call'}
//List of stations before this station
PROPERTY StationsAhead : I_CH_List
GET
StationsAhead := THIS^.fbStationsAhead;
END_GET
END_PROPERTY

{attribute 'monitoring':='call'}
//List of stations behinde this station
PROPERTY StationsBehinde : I_CH_List
GET
StationsBehinde := THIS^.fbStationsBehinde;
END_GET
END_PROPERTY

METHOD Update : HRESULT
VAR_INST
	nCtsDebug : UINT;
END_VAR
VAR
	ipFirstMoverInQueue: I_XP_Mover;
	//ipFirstMoverInQueuePlc : I_XP_Mover_PLC;
	ipFirstMoverInQueueObj : I_CH_Object;
	iStation: I_XP_Station;
	stPath: ST_PathFinder_1;
	bValideStationToStartMove : BOOL;
	bThisStationAsTarged : BOOL;
	
	ipThisStation : I_XP_Station := THIS^;
	
	//bNotThisStationAsTarged : BOOL;
	bMoverValideToSendAway : BOOL;
	bInReachForNewCmd : BOOL;
	bThisStationAsParent : BOOL;
	sTargedStation : STRING;
	ipPath : I_XP_Path;
	ipMover : I_XP_Mover;
END_VAR
//Force to do init befor call update
IF NOT bInitDone THEN
	THIS^.Initialize();
	RETURN;
END_IF

THIS^.Prepare();//Prepare time-critical information, if not already done


// ********************** Set feedback depending on active command *******************************
IF THIS^.eActiveCommand <> E_NcAxisCommands.None THEN
	fbFeedback.ActiveCommand 	:= TO_STRING(THIS^.eActiveCommand);	
END_IF

CASE THIS^.eActiveCommand OF

	E_NcAxisCommands.Initialize:
		fbFeedback.Busy 			:= NOT THIS^.bInitDone;
		fbFeedback.Done 			:= THIS^.bInitDone;
		fbFeedback.ErrorId 			:= 0;
		                        	

	ELSE//External command in subclass
		;
END_CASE


// **********************  Stop to execute commands on .done or .error ***************************
IF fbFeedback.Done OR THIS^.fbFeedback.Error THEN
	eActiveCommand 				:= E_NcAxisCommands.None;
END_IF



// If enabled start station logic
IF THIS^.ipXpSystem.Enabled THEN
	
	// Process Simulation. All functionality packed into one method for easier overwriting
	THIS^.Simulation();


	
	//Detect mover who is passing the station whitout be in queue. Adjust to new Gap
	IF fbTrigger.MoverDetected AND (fbTrigger.MoverAtTrigger <> 0) AND NOT THIS^.bSuppressDynamicsChange THEN
		//Only if not in this queue
		IF fbTrigger.MoverAtTrigger.ParentStation <> ipThisStation THEN
			fbTrigger.MoverAtTrigger.MoveOnTrack(ipTrack	:= fbTrigger.MoverAtTrigger.LastCmdTargedTrack,
												fPosition	:= fbTrigger.MoverAtTrigger.LastCmdTargedPosition, 
												fGap		:= THIS^.fMoverGapAtExit);
		END_IF
	END_IF	
	
	
	
	//Test if the first mover is in station and send him away, if the destination is not this station	
	IF __QUERYINTERFACE(THIS^.MoversInQueue[0],ipFirstMoverInQueue) THEN
		bThisStationAsTarged := (ipFirstMoverInQueue.TargetStation = THIS^.TargetGroupe) OR (ipFirstMoverInQueue.TargetStation = THIS^.LUID); 
		bThisStationAsParent := ipFirstMoverInQueue.ParentStation.LUID = THIS^.LUID;
		bInReachForNewCmd	:= ipFirstMoverInQueue.DistToParentStation <= XPlanarParameterlist.F_DIST_SET_NEW_MOVE_CMD_BEFORE_REACHING_PARENT_STATION;
		
	//	bNotThisStationAsTarged := NOT bThisStationAsTarged; 
	//	bMoverValideToSendAway := bNotThisStationAsTarged AND (ipFirstMoverInQueue.DistToParentStation <= XPlanarParameterlist.F_DIST_SET_NEW_MOVE_CMD_BEFORE_REACHING_PARENT_STATION);
	
	END_IF
	IF ipFirstMoverInQueue = 0 OR NOT bInReachForNewCmd THEN
		; //Do Nothing, no mover
	

	ELSIF bThisStationAsTarged THEN
		;//Do Nothing, wait for proccess

		
	ELSIF bThisStationAsParent THEN
		//Get a path to a new parent or targed
		sTargedStation := ipFirstMoverInQueue.TargetStation;
		stPath := THIS^.searchNextBestStationByName(sTargedStation := sTargedStation, nPermittedSearchDepth := XPlanarParameterlist.N_MAX_SEARCH_DEPTH, bCallFromExternal:=TRUE);
		
		bValideStationToStartMove := stPath.bTargetFound AND (stPath.ipBestStation <> 0);
		//Start Movement
		IF bValideStationToStartMove THEN 
			
			nCtsDebug := nCtsDebug +1;
			
			ipFirstMoverInQueue.Route.Duplicate(stPath.ipRouteToParent);
		
			//deregister from this station and register with a new parrent station
			ipFirstMoverInQueueObj := THIS^.fbAssignedMovers.FindOID(ipFirstMoverInQueue.OID);
			THIS^.fbAssignedMovers.RemoveObject(ipFirstMoverInQueueObj);
			stPath.ipBestStation.AddMoverToQueue(ipFirstMoverInQueue);	

 		END_IF     
	END_IF
	
	
	//check all movers if this station is a start of an path	
	ipXpSystem.Movers.ResetIterator();
	WHILE ipXpSystem.Movers.HasNextObject() DO
		IF __QUERYINTERFACE(ipXpSystem.Movers.GetNextObject(),ipFirstMoverInQueue) AND_THEN ipFirstMoverInQueue.CurrentTrack = ipThisStation.AccocietedTrack AND_THEN (ABS(ipFirstMoverInQueue.PositionOnTrack - ipThisStation.PositionOnTrack) < THIS^.fDecisionDistance) THEN
			ipFirstMoverInQueue.Route.ResetIterator();
			WHILE ipFirstMoverInQueue.Route.HasNextObject() DO
				IF __QUERYINTERFACE(ipFirstMoverInQueue.Route.GetNextObject(), ipPath) AND_THEN ipPath.StationStart = ipThisStation THEN
					//Remove this path from route and send to path desination
					ipFirstMoverInQueue.Route.RemoveObject(ipPath);
						
					
					//If mover is standstill in current station, send him away whit the exit gap, else use the in mover stored gap
					IF LREAL_TO_DINT(ipFirstMoverInQueue.PositionOnTrack) = LREAL_TO_DINT(THIS^.PositionOnTrack) THEN
						ipFirstMoverInQueue.MoveOnTrackToStation(ipStation := ipPath.StationDestination,
													fGap:= THIS^.fMoverGapAtExit);					
					ELSE
						ipFirstMoverInQueue.MoveOnTrackToStation(ipStation := ipPath.StationDestination,
													fGap:= ipFirstMoverInQueue.LastCmdTargedGap);
					END_IF	
				END_IF
			END_WHILE
			ipFirstMoverInQueue.Route.RestoreIterator();
		END_IF		
	END_WHILE
	ipXpSystem.Movers.RestoreIterator();
END_IF



Update := S_OK;
END_METHOD

END_FUNCTION_BLOCK

// COMPONENTs/Stationen/I_XP_Station_PLC
INTERFACE I_XP_Station_PLC EXTENDS __SYSTEM.IQueryInterface

{attribute 'monitoring':='call'}
PROPERTY CtsEmptySpaceInQueue : UDINT
GET
END_GET
END_PROPERTY

{attribute 'monitoring':='call'}
PROPERTY CtsMoversInQueue : UDINT
GET
END_GET
END_PROPERTY

{attribute 'monitoring':='call'}
PROPERTY LUID : STRING //Locally unique identifier
GET
END_GET
END_PROPERTY

{attribute 'monitoring':='call'}
PROPERTY MoverQueueSize : UINT
GET
END_GET
SET
END_SET
END_PROPERTY

{attribute 'monitoring':='call'}
PROPERTY MoversInPlace : BOOL
GET
END_GET
END_PROPERTY

{attribute 'monitoring':='call'}
PROPERTY MoversInQueue : REFERENCE TO ARRAY [0..(CHALET_BaseComponents.BaseParameterlist.MAX_OBJECTS-1)] OF I_XP_Mover_PLC // Return a sorted list of movers in this zone. Index 0 is the mover in Front
GET
END_GET
END_PROPERTY

{attribute 'monitoring':='call'}
//prevent further movers from entering the station, 
//e.g. to prevent a collision. All movers that are already moving to reach this station will be stopped with a stop 
//and restarted with Ready True.
PROPERTY ReadyToRecvMovers : BOOL
GET
END_GET
SET
END_SET
END_PROPERTY

METHOD SendMoversToStation : I_CH_Feedback //All movers in the station are sent to this destination
VAR_INPUT
	sTargetStation: STRING;//unique station name or group of stations
END_VAR
END_METHOD

{attribute 'monitoring':='call'}
//A time that is waited as soon as the mover is in the station (including the monitoring window) before “MoversInPlace” is set. e.g. used to stabilize the workpiece
PROPERTY TargetPosMonitoringTime : TIME
GET
END_GET
SET
END_SET
END_PROPERTY

{attribute 'monitoring':='call'}
//How many mm before the mover reaches the position is “MoversInPlace” set for the process. 
//This distance can also be set very large (e.g. 100mm) for moving past without stopping.
PROPERTY TargetPosWindow : LREAL
GET
END_GET
SET
END_SET
END_PROPERTY

{attribute 'monitoring':='call'}
PROPERTY ProcessSimulationActive : BOOL
GET
END_GET
END_PROPERTY

//If a valid time (>0seconds) is set and the configured destination station exists, then the movers will be sent away automatically after this time from now on.
METHOD SimulationMode : HRESULT
VAR_INPUT
	fProcessDuration 		: LREAL; //[s]
	sTargedStation	: STRING; //Group of the targed station to automatic send after the duration
END_VAR
END_METHOD

{attribute 'monitoring':='call'}
//Track on which the station is located
PROPERTY AccocietedTrack : I_XP_Track
GET
END_GET
END_PROPERTY

{attribute 'monitoring':='call'}
PROPERTY Feedback : I_CH_Feedback
GET
END_GET
END_PROPERTY

{attribute 'monitoring':='call'}
//Filter content, movers with one of these targets may not approach or drive over the station
PROPERTY Filter : STRING
GET
END_GET
SET
END_SET
END_PROPERTY

{attribute 'monitoring':='call'}
PROPERTY MoverGapAtExit : LREAL //[mm] Every mover that leaves or passes the station gets this new gap as a target.
GET
END_GET
SET
END_SET
END_PROPERTY

{attribute 'monitoring':='call'}
//[mm] from the beginning of the assigned track
PROPERTY PositionOnTrack : LREAL
GET
END_GET
END_PROPERTY

{attribute 'monitoring':='call'}
//Position on the assigned track
PROPERTY PositionOnTrackXY : REFERENCE TO PositionXY
GET
END_GET
END_PROPERTY

{attribute 'monitoring':='call'}
//Planned position, not necessarily on the track
PROPERTY PositionXY : REFERENCE TO  PositionXY
GET
END_GET
END_PROPERTY

{attribute 'monitoring':='call'}
//List of stations before this station
PROPERTY StationsAhead : I_CH_List
GET
END_GET
END_PROPERTY

{attribute 'monitoring':='call'}
//List of stations behinde this station
PROPERTY StationsBehinde : I_CH_List
GET
END_GET
END_PROPERTY

{attribute 'monitoring':='call'}
PROPERTY TargetGroupe : STRING
GET
END_GET
END_PROPERTY

END_INTERFACE

// COMPONENTs/System/I_XP_System_PLC
INTERFACE I_XP_System_PLC EXTENDS I_CH_Object

METHOD CheckTargetExists : BOOL //Return TRUE if target is existing
VAR_INPUT
	sStation	: STRING; //Group of the targed station or LUID
END_VAR
END_METHOD

METHOD Disable : I_CH_Feedback
VAR_INPUT
END_VAR
END_METHOD

{attribute 'monitoring':='call'}
PROPERTY Disabled : BOOL
GET
END_GET
END_PROPERTY

METHOD Enable : I_CH_Feedback
VAR_INPUT
END_VAR
END_METHOD

{attribute 'monitoring':='call'}
PROPERTY Enabled : BOOL
GET
END_GET
END_PROPERTY

{attribute 'monitoring':='call'}
PROPERTY Enviroment : I_XP_Environment
GET
END_GET
END_PROPERTY

{attribute 'monitoring':='call'}
PROPERTY Feedback : CHALET_BaseComponents.I_CH_Feedback
GET
END_GET
END_PROPERTY

METHOD Initialize : HRESULT
VAR_INPUT
END_VAR
END_METHOD

{attribute 'monitoring':='call'}
PROPERTY Initialized : BOOL
GET
END_GET
END_PROPERTY

{attribute 'monitoring':='call'}
PROPERTY Movers : CHALET_BaseComponents.I_CH_LIST
GET
END_GET
END_PROPERTY

METHOD Station : I_XP_Station_PLC
VAR_INPUT
	sLUID : STRING;
END_VAR
END_METHOD

{attribute 'monitoring':='call'}
PROPERTY Stations : CHALET_BaseComponents.I_CH_LIST
GET
END_GET
END_PROPERTY

{attribute 'monitoring':='call'}
PROPERTY Tracks : CHALET_BaseComponents.I_CH_LIST
GET
END_GET
END_PROPERTY

{attribute 'monitoring':='call'}
PROPERTY Triggers : CHALET_BaseComponents.I_CH_LIST
GET
END_GET
END_PROPERTY

METHOD Update : HRESULT
VAR_INPUT
END_VAR
END_METHOD

{attribute 'monitoring':='call'}
PROPERTY Zones : CHALET_BaseComponents.I_CH_LIST
GET
END_GET
END_PROPERTY

END_INTERFACE

// COMPONENTs/System/FB_XP_System
{attribute 'no_explicit_call' := 'Do not call the body - Stick to OOP'}
(* XPlanar System - 1 per associated XPlanar 
	The system is the container and organizer for all subsequent XPlanar objects. All objects are registered with this system*)
FUNCTION_BLOCK FB_XP_System EXTENDS FB_CH_Object IMPLEMENTS I_XP_System_Registration, I_XP_System_PLC
VAR	
	{attribute 'hide'}
	bInitDone : BOOL;
	{attribute 'hide'}
	bErrorDuringFbInit : BOOL; // Not possible to reset
	{attribute 'hide'}                   	
	eActiveCommand 		: CHALET_Nc.E_NcAxisCommands := CHALET_Nc.E_NcAxisCommands.None;
	{attribute 'hide'}
    fbMovers     : FB_CH_List;
	{attribute 'hide'}	
    fbTracks     : FB_CH_List;
	{attribute 'hide'}	
	fbStations 	 : FB_CH_List;
	{attribute 'hide'}	
	fbTriggers 	 : FB_CH_List;
	{attribute 'hide'}	
	fbZones 	 : FB_CH_List;
	{attribute 'hide'}	
    ipGroup       : I_XP_Group;
	{attribute 'hide'}	
    ipEnvironment : I_XP_Environment;
	{attribute 'hide'}
    nSeqEnabling  : UINT;
	{attribute 'hide'}
	nSeqJoiningTrack : UINT;
	{attribute 'hide'}
	nSeqJoiningStation : UINT;
	{attribute 'hide'}	
    nSeqDisabling  : UINT := SEQ_DONE;
	{attribute 'hide'}
	fbFeedback : FB_CH_Feedback;
	
	//ZZZ TODO this port is not fix. REad from the task object
	nXPlanarTaskAdsPort : UINT;
END_VAR
VAR CONSTANT
	{attribute 'hide'}
	SEQ_DONE : UINT := 999;
END_VAR

METHOD PROTECTED JoiningStation : HRESULT
VAR
	hr : HRESULT;
	ipEachMover : I_XP_Mover;
	ipEachMoverPlc : I_XP_Mover_PLC;
	ipEachMoverInStation : I_XP_Mover;
	ipEachStation : I_XP_Station;
	ipFirstStation : I_XP_Station;
	ipParentStation : I_XP_Station;
	ipTempMoverPlc : I_XP_Mover_PLC;
	
	//during move on track
	fVelo, fAccDec	: Tc3_Mc3Definitions.MC_LREAL := Tc3_Mc3Definitions.MC_DEFAULT;
END_VAR
VAR_INST
	{attribute 'hide'}	
	fbDelayJoiningStation : TON;
END_VAR
CASE nSeqJoiningStation OF

	0: //Init
		fbDelayJoiningStation.IN := FALSE;
		nSeqJoiningStation := 10;
	
		
	10:	//Distribute the movers to the available stations.
		(*Send the movers to the last assigned station:
		  For this purpose, the list of assigned movers is checked at each station and the mover is given a new move command to the station.
		  If there are still movers in the system that do not have a move command, these are sent to station 1. Typically after starting up
		  *)
		
		//Do for each mover in a station
		THIS^.fbStations.ResetIterator();    
		WHILE THIS^.fbStations.HasNextObject() DO
			ToXpStation(THIS^.fbStations.GetNextObject(),ipEachStation);
				//Do for all in station assigned Movers
				ipEachStation.AssignedMovers.ResetIterator();
				WHILE ipEachStation.AssignedMovers.HasNextObject() DO
					ToXpMover(ipEachStation.AssignedMovers.GetNextObject(),ipEachMoverInStation);
					//Send to assigned station - Shortest way
					hr := GetMostSignificant(hr, ipEachMoverInStation.MoveOnTrack_ShortestWay(ipTrack	:= ipEachStation.AccocietedTrack, 
																							  fPosition	:= ipEachStation.PositionOnTrack,
																							  fGap 		:= ipEachMoverInStation.LastCmdTargedGap));
				END_WHILE
		END_WHILE        
		nSeqJoiningStation := 20;
		
	20:	//Test if there is an Mover whitout an active TargedStation (first startup)
		//Send them to first station
		THIS^.fbStations.ResetIterator();
		IF THIS^.fbStations.HasNextObject() THEN
			//Get interface to first Station in list
			ToXpStation(THIS^.fbStations.GetNextObject(),ipFirstStation);
			//Set as targed station the first station in list. but as the parent the station in front of the first one(if existing) 
			//(the parent station is not necessarily the target station. But the station that is responsible for sending the mover forward if necessary)
			ipFirstStation.StationsAhead.ResetIterator();
			ToXpStation(ipFirstStation.StationsAhead.GetNextObject(),ipParentStation);
			
			//Check for mover whitout a targed station
			THIS^.fbMovers.ResetIterator();
			WHILE THIS^.fbMovers.HasNextObject() DO
				//Do for all Movers whitout a targed station
				IF ToXpMover(THIS^.fbMovers.GetNextObject(),ipEachMover) AND_THEN (ipEachMover.TargetStation = '') AND_THEN __QUERYINTERFACE(ipEachMover,ipEachMoverPlc) THEN
					//Set Path dynamic constraint to settings in XPlanarParameterlist. 0=Defalt
					IF XPlanarParameterlist.F_ENABLING_ON_TRACK_VELOCITY <> 0 THEN fVelo := XPlanarParameterlist.F_ENABLING_ON_TRACK_VELOCITY;END_IF
					IF XPlanarParameterlist.F_ENABLING_ON_TRACK_ACC_DEC <> 0 THEN fAccDec := XPlanarParameterlist.F_ENABLING_ON_TRACK_ACC_DEC;END_IF
				
					//Increase or decrease the mover DynConstraint for approaching the station 
					ipEachMoverPlc.SetDynConstraint_Path(	V:= fVelo, 
															A:= fAccDec, 
															D:= fAccDec, 
															J:= Tc3_Mc3Definitions.MC_DEFAULT);
		
					//Set as targed station the first station in list. but as the parent the station in front of the first one(if existing) 
					IF ipParentStation <> 0 THEN
						hr := GetMostSignificant(hr, ipEachMover.MoveOnTrackToStation(ipParentStation, XPlanarParameterlist.F_GAP_STARTUP));
						hr := GetMostSignificant(hr, ipParentStation.AddMoverToQueue(ipEachMover));
						ipEachMover.TargetStation := ipFirstStation.TargetGroupe;
					ELSE
						//If no partent station is existing
						hr := GetMostSignificant(hr, ipEachMover.MoveOnTrackToStation(ipFirstStation, XPlanarParameterlist.F_GAP_STARTUP));
						hr := GetMostSignificant(hr, ipFirstStation.AddMoverToQueue(ipEachMover));
						ipEachMover.TargetStation := ipFirstStation.TargetGroupe;
					END_IF
					
					
					//Set Path dynamic constraint back to default
					ipEachMoverPlc.SetDynConstraint_Path(	V:= Tc3_Mc3Definitions.MC_DEFAULT, 
															A:= Tc3_Mc3Definitions.MC_DEFAULT, 
															D:= Tc3_Mc3Definitions.MC_DEFAULT, 
															J:= Tc3_Mc3Definitions.MC_DEFAULT);
		
				END_IF
			END_WHILE
		END_IF

		nSeqJoiningStation := 30;
		
	30: //Delay to allow the movers to start movement
		fbDelayJoiningStation.IN := TRUE;
		fbDelayJoiningStation.PT := T#2S;
		IF fbDelayJoiningStation.Q THEN
			nSeqJoiningStation := 40;
			fbDelayJoiningStation.IN := FALSE;
		END_IF
	
	
	40: //Wait for all movers until the movement is completed(speed =0)
		THIS^.fbMovers.ResetIterator();
		WHILE THIS^.fbMovers.HasNextObject() DO
			IF ToXpMover(THIS^.fbMovers.GetNextObject(),ipEachMover) THEN
				//Check all movers if an error is active
				IF ipEachMover.Feedback.Error THEN
					hr := GetMostSignificant(hr, ipEachMover.Feedback.HR);
				//Wait for all movers to stop/finish movement
				ELSIF NOT (ipEachMover.PlanarMover.MCTOPLC.SETONTRACK.SetVelo = 0.0) THEN
					hr := GetMostSignificant(hr, S_PENDING);
				END_IF
			END_IF
		END_WHILE
		
		IF CheckOk(hr) THEN 
			nSeqJoiningStation := SEQ_DONE;
		ELSIF FAILED(hr) THEN
			nSeqJoiningStation := 1000 + nSeqJoiningStation;
		END_IF			

	
	1000..1999://Error
		hr := GetMostSignificant(hr, E_FAIL);
END_CASE

//Update
fbDelayJoiningStation();


//Return value
IF FAILED(hr) THEN 
	//Error
    JoiningStation := GetMostSignificant(hr, E_FAIL);
ELSIF (nSeqJoiningStation = SEQ_DONE) THEN
	//Done
    JoiningStation := S_OK;
ELSE
	//Busy
    JoiningStation := S_PENDING;;
END_IF
END_METHOD

METHOD PROTECTED JoiningTrack : HRESULT
VAR	
	hr : HRESULT;
	ipClosestTrack : I_XP_Track;	
	ipEachMover : I_XP_Mover;
	ipEachTrack : I_XP_Track;
	fDistance : LREAL;
	fShortestDistance : LREAL;
END_VAR
CASE nSeqJoiningTrack OF

	0: //Init
		nSeqJoiningTrack := 10;
	
		
	
	10:// Join closest track
		THIS^.fbMovers.ResetIterator();
		WHILE THIS^.fbMovers.HasNextObject() DO
			IF ToXpMover(THIS^.fbMovers.GetNextObject(),ipEachMover) THEN
				
				//check all track to decide which is the closest
				THIS^.fbTracks.ResetIterator();
				//start with the greatest possible distance, so that each track is definitely closer
				fShortestDistance := CHALET_BaseComponents.GVL_Datatypes.cMaxLreal; 
				WHILE THIS^.fbTracks.HasNextObject() DO
					IF ToXpTrack(THIS^.fbTracks.GetNextObject(),ipEachTrack) THEN
						fDistance := ipEachMover.DistToTrack(ipEachTrack);
						//closer track found
						IF fDistance <= fShortestDistance THEN
							ipClosestTrack := ipEachTrack;
							fShortestDistance := fDistance;
						END_IF
					END_IF
				END_WHILE
				
				//send mover to found closest track
				IF ipClosestTrack <> 0 THEN
					hr := GetMostSignificant(hr, ipEachMover.JoinTrack(ipClosestTrack));
				ELSE
					hr := GetMostSignificant(hr, E_FAIL);
				END_IF
			END_IF
		END_WHILE
		nSeqJoiningTrack := 20;
		
		
	20: // Joining closest track check feedback
		IF NOT fbTracks.IsEmpty THEN
			THIS^.fbMovers.ResetIterator();
			WHILE THIS^.fbMovers.HasNextObject() DO
				IF ToXpMover(THIS^.fbMovers.GetNextObject(),ipEachMover) THEN
					
					// Check mover errors
					hr := GetMostSignificant(hr, ipEachMover.Feedback.HR);
					
					//Check if Mover is on track
					IF NOT (ipEachMover.Mode = MC_PLANAR_MOVER_COMMAND_MODE.OnTrack) THEN
						hr := GetMostSignificant(hr, S_PENDING);
					END_IF
				END_IF
			END_WHILE
		END_IF
		
		IF CheckOk(hr) THEN 
			nSeqJoiningTrack := SEQ_DONE;
		ELSIF FAILED(hr) THEN
			nSeqJoiningTrack := 1000 + nSeqJoiningTrack;
		END_IF			

		
	1000..1999://Error
		hr := GetMostSignificant(hr, E_FAIL);
END_CASE

		
		
//Return value
IF FAILED(hr) THEN 
	//Error
    JoiningTrack := GetMostSignificant(hr, E_FAIL);
ELSIF (nSeqJoiningTrack = SEQ_DONE) THEN
	//Done
    JoiningTrack := S_OK;
ELSE
	//Busy
    JoiningTrack := S_PENDING;;
END_IF
END_METHOD

METHOD Disable : I_CH_Feedback
VAR_INPUT
END_VAR
//Disable is allways posible

THIS^.nSeqDisabling 	:= 1;
THIS^.nSeqEnabling 		:= 0;

THIS^.eActiveCommand 				:= CHALET_NC.E_NcAxisCommands.Disable;
THIS^.fbFeedback.LastCommandAccepted:= TRUE;		
THIS^.fbFeedback.Busy 				:= TRUE;
		
Disable := THIS^.fbFeedback;
END_METHOD

{attribute 'monitoring':='call'}
PROPERTY Disabled : BOOL
GET
Disabled := nSeqDisabling = SEQ_DONE OR 
			(nSeqDisabling = 0 AND nSeqEnabling = 0);
END_GET
END_PROPERTY

METHOD PROTECTED Disabling : HRESULT
VAR
	hr : HRESULT;
	bOk : BOOL := TRUE;
	iTempMover : I_XP_Mover;
	iTempTrack : I_XP_Track;
END_VAR
VAR_INST
	hrLastCycle : HRESULT;
END_VAR
Disabling := S_PENDING;
CASE nSeqDisabling OF
	0: // Idle
		Disabling := S_OK;
		
		
	1: // Halt movers
		THIS^.fbMovers.ResetIterator();
		WHILE THIS^.fbMovers.HasNextObject() DO
			IF ToXpMover(THIS^.fbMovers.GetNextObject(),iTempMover) THEN
				hr := GetMostSignificant(hr, iTempMover.Halt());
			END_IF
		END_WHILE
		
		IF CheckOk(hr) THEN 
			nSeqDisabling := 20;
		ELSE
			nSeqDisabling := 1000 + nSeqDisabling;
		END_IF	
	
		
	20: // Halting movers
		THIS^.fbMovers.ResetIterator();
		WHILE THIS^.fbMovers.HasNextObject() DO
			IF ToXpMover(THIS^.fbMovers.GetNextObject(),iTempMover) THEN
				bOk := bOk AND iTempMover.PlanarMover.MCTOPLC.SET.SetVelo.x = 0;
				bOk := bOk AND iTempMover.PlanarMover.MCTOPLC.SET.SetVelo.y = 0;
				bOk := bOk AND iTempMover.PlanarMover.MCTOPLC.SET.SetVelo.z = 0;
				bOk := bOk AND iTempMover.PlanarMover.MCTOPLC.SET.SetVelo.a = 0;
				bOk := bOk AND iTempMover.PlanarMover.MCTOPLC.SET.SetVelo.b = 0;
				bOk := bOk AND iTempMover.PlanarMover.MCTOPLC.SET.SetVelo.c = 0;
			END_IF
		END_WHILE
		
		IF bOk THEN 
			nSeqDisabling := 30;
		END_IF	
		
	
	30: // Reset movers
		THIS^.fbMovers.ResetIterator();
		WHILE THIS^.fbMovers.HasNextObject() DO
			IF ToXpMover(THIS^.fbMovers.GetNextObject(),iTempMover) THEN
				hr := GetMostSignificant(hr, iTempMover.Reset());
			END_IF
		END_WHILE
		
		IF CheckOk(hr) THEN 
			nSeqDisabling := 40;
		ELSE
			nSeqDisabling := 1000 + nSeqDisabling;
		END_IF		
		
		
	40: // Resetting movers
		THIS^.fbMovers.ResetIterator();
		WHILE THIS^.fbMovers.HasNextObject() DO
			IF ToXpMover(THIS^.fbMovers.GetNextObject(),iTempMover) THEN
				hr := GetMostSignificant(hr, iTempMover.Feedback.HR);
			END_IF
		END_WHILE
		
		IF CheckOk(hr) THEN 
			nSeqDisabling := 50;
		ELSIF FAILED(hr) THEN
			nSeqDisabling := 1000 + nSeqDisabling;
		END_IF
		
		
	50: // Disable movers
		THIS^.fbMovers.ResetIterator();
		WHILE THIS^.fbMovers.HasNextObject() DO
			IF ToXpMover(THIS^.fbMovers.GetNextObject(),iTempMover) THEN
				hr := GetMostSignificant(hr, iTempMover.Disable());
			END_IF
		END_WHILE
		
		IF CheckOk(hr) THEN 
			nSeqDisabling := 60;
		ELSE
			nSeqDisabling := 1000 + nSeqDisabling;
		END_IF			
		
		
	60: // Disabling movers
		THIS^.fbMovers.ResetIterator();
		WHILE THIS^.fbMovers.HasNextObject() DO
			IF ToXpMover(THIS^.fbMovers.GetNextObject(),iTempMover) THEN
				hr := GetMostSignificant(hr, iTempMover.Feedback.HR);
			END_IF
		END_WHILE
		
		IF CheckOk(hr) THEN 
			nSeqDisabling := 61;
		ELSIF FAILED(hr) THEN
			nSeqDisabling := 1000 + nSeqDisabling;
		END_IF		


	61: // Reset track
		THIS^.fbTracks.ResetIterator();
		WHILE THIS^.fbTracks.HasNextObject() DO
			IF ToXpTrack(THIS^.fbTracks.GetNextObject(),iTempTrack) THEN
				hr := GetMostSignificant(hr, iTempTrack.Reset());
			END_IF
		END_WHILE
		
		IF CheckOk(hr) THEN 
			nSeqDisabling := 62;
		ELSE
			nSeqDisabling := 1000 + nSeqDisabling;
		END_IF		
		
		
	62: // Resetting track
		THIS^.fbTracks.ResetIterator();
		WHILE THIS^.fbTracks.HasNextObject() DO
			IF ToXpTrack(THIS^.fbTracks.GetNextObject(),iTempTrack) THEN
				hr := GetMostSignificant(hr, iTempTrack.Feedback.HR);
			END_IF
		END_WHILE
		
		IF CheckOk(hr) THEN 
			nSeqDisabling := 63;
		ELSIF FAILED(hr) THEN
			nSeqDisabling := 1000 + nSeqDisabling;
		END_IF	

				
	63: // Reset group
		hr := ipGroup.Reset();
		
		IF CheckOk(hr) THEN 
			nSeqDisabling := 64;
		ELSE
			nSeqDisabling := 1000 + nSeqDisabling;
		END_IF		
		
		
	64: // Resetting group
		hr := ipGroup.Feedback.HR;
		
		IF CheckOk(hr) THEN 
			nSeqDisabling := 70;
		ELSIF FAILED(hr) THEN
			nSeqDisabling := 1000 + nSeqDisabling;
		END_IF		
		
		
		

   70: // Disable tracks
		THIS^.fbTracks.ResetIterator();
		WHILE THIS^.fbTracks.HasNextObject() DO
			IF ToXpTrack(THIS^.fbTracks.GetNextObject(),iTempTrack) THEN
				hr := GetMostSignificant(hr, iTempTrack.Disable());
			END_IF
		END_WHILE
		
		IF CheckOk(hr) THEN 
			nSeqDisabling := 80;
		ELSE
			nSeqDisabling := 1000 + nSeqDisabling;
		END_IF			
   
		
   80: // Disabling tracks
		THIS^.fbTracks.ResetIterator();
		WHILE THIS^.fbTracks.HasNextObject() DO
			IF ToXpTrack(THIS^.fbTracks.GetNextObject(),iTempTrack) THEN
				hr := GetMostSignificant(hr, iTempTrack.Feedback.HR);
			END_IF
		END_WHILE
		
		IF CheckOk(hr) THEN 
			nSeqDisabling := 90;
		ELSIF FAILED(hr) THEN
			nSeqDisabling := 1000 + nSeqDisabling;
		END_IF	
				

	90: // Disable group
		hr := ipGroup.Disable();
		
		IF CheckOk(hr) THEN 
			nSeqDisabling := 100;
		ELSE
			nSeqDisabling := 1000 + nSeqDisabling;
		END_IF	
		
		
   100: // Disabling group
		hr := ipGroup.Feedback.HR;
		
		IF CheckOk(hr) THEN 
			nSeqDisabling := 105;
		ELSIF FAILED(hr) THEN
			nSeqDisabling := 1000 + nSeqDisabling;
		END_IF	

		
  105: // Remove tracks from group
		THIS^.fbTracks.ResetIterator();
		WHILE THIS^.fbTracks.HasNextObject() DO
			IF ToXpTrack(THIS^.fbTracks.GetNextObject(),iTempTrack) THEN
				hr := GetMostSignificant(hr, iTempTrack.RemoveFromGroup());
			END_IF
		END_WHILE
		
		IF CheckOk(hr) THEN 
			nSeqDisabling := 106;
		ELSE
			nSeqDisabling := 1000 + nSeqDisabling;
		END_IF			
   
		
   106: // Removing tracks from group
		THIS^.fbTracks.ResetIterator();
		WHILE THIS^.fbTracks.HasNextObject() DO
			IF ToXpTrack(THIS^.fbTracks.GetNextObject(),iTempTrack) THEN
				bOk := bOk AND iTempTrack.PlanarTrack.MCTOPLC_STD.GroupOID = 0;
			END_IF
		END_WHILE
		
		IF bOk THEN 
			nSeqDisabling := 110;
		END_IF	
		
		
	110: // Remove movers from group
		THIS^.fbMovers.ResetIterator();
		WHILE THIS^.fbMovers.HasNextObject() DO
			IF ToXpMover(THIS^.fbMovers.GetNextObject(),iTempMover) THEN
				hr := GetMostSignificant(hr, iTempMover.RemoveFromGroup());
			END_IF
		END_WHILE
		
		IF CheckOk(hr) THEN 
			nSeqDisabling := 120;
		ELSE
			nSeqDisabling := 1000 + nSeqDisabling;
		END_IF		
	
		
	120: // Removing movers from group
		THIS^.fbMovers.ResetIterator();
		WHILE THIS^.fbMovers.HasNextObject() DO
			IF ToXpMover(THIS^.fbMovers.GetNextObject(),iTempMover) THEN
				bOk := bOk AND iTempMover.PlanarMover.MCTOPLC.STD.GroupOID = 0;
			END_IF
		END_WHILE
		
		IF bOk THEN 
			nSeqDisabling := 130;
		END_IF		
	
		
	130: // Remove envirement from group
		hr := ipEnvironment.RemoveFromGroup();
		
		IF CheckOk(hr) THEN 
			nSeqDisabling := 140;
		ELSE
			nSeqDisabling := 1000 + nSeqDisabling;
		END_IF		
		
		
   140: // Removing envirement from group
		//IF CheckOk(iEnvironment.HR) OR (iEnvironment.Self.MCTOPLC_STD.GroupOID = 0) THEN 
		hr := ipEnvironment.Feedback.HR;
	
		IF CheckOk(hr) THEN 
			nSeqDisabling := SEQ_DONE;
		ELSIF FAILED(hr) THEN
			nSeqDisabling := 1000 + nSeqDisabling;
		END_IF	
		
	
   SEQ_DONE: //Done
   		Disabling := S_OK;

		
	1000..1999://Error
		hr := GetMostSignificant(hrLastCycle, E_FAIL);

END_CASE

//store last information
hrLastCycle := hr;

// Propagate error
IF FAILED(hr) THEN
	Disabling := hr;
END_IF
END_METHOD

METHOD Enable : CHALET_BaseComponents.I_CH_Feedback
VAR_INPUT
END_VAR
IF NOT THIS^.fbFeedback.Done THEN
	//Error active/not ready
	THIS^.fbFeedback.LastCommandAccepted 	:= FALSE;

ELSIF nSeqEnabling <> 0 THEN
	//System is partial or full enabled. Disable first.
	THIS^.fbFeedback.LastCommandAccepted 	:= FALSE;
ELSE
	THIS^.nSeqDisabling 	:= 0;
	THIS^.nSeqEnabling 		:= 1;
	
	THIS^.eActiveCommand 				:= CHALET_NC.E_NcAxisCommands.Enable;
	THIS^.fbFeedback.LastCommandAccepted:= TRUE;		
	THIS^.fbFeedback.Busy 				:= TRUE;	
END_IF

Enable := THIS^.fbFeedback;
END_METHOD

{attribute 'monitoring':='call'}
PROPERTY Enabled : BOOL
GET
Enabled := nSeqEnabling = SEQ_DONE;
END_GET
END_PROPERTY

METHOD PROTECTED Enabling : HRESULT
VAR
	hr : HRESULT;
	bWatchDogActive : BOOL;
	
	ipTempMover : I_XP_Mover;
	ipTempMoverPlc : I_XP_Mover_PLC;
	ipTempStation : I_XP_Station;
	ipTempTrack : I_XP_Track;
	
	lrCRotationShortestPos : LREAL;
	
	nSupSeq : UINT;
END_VAR

VAR_INST
	fbTimeOutSeq : TON; 
	hrLastCycle 	: HRESULT;
	nlastState	: UINT;
	
	{attribute 'hide'}	
	fbTimeOutEnabling : FB_TcAlarm;
	{attribute 'hide'}	
	fbErrorEnabling : FB_TcAlarm;
END_VAR
Enabling := S_PENDING;
CASE nSeqEnabling OF
	0: // Idle
		Enabling := S_OK;	
		
	1: //Redetect all movers on real system
		bWatchDogActive := TRUE;
		IF THIS^.ipEnvironment.UtilityEnvirement.XpuTcIo(1).GetOperationMode() = OperationMode.Normal THEN
			THIS^.ipEnvironment.UtilityEnvirement.XpuTcIo(1).SetStartMoverRedetection();	
		END_IF
		nSeqEnabling := 5;

		
	5: //Compare detectet and expectet movers	
	   //timeout is monitored in this sequence
		bWatchDogActive := TRUE;
		IF (THIS^.ipEnvironment.UtilityEnvirement.XpuTcIo(1).GetMoverDetectionInfos().APM4220Detected = THIS^.ipEnvironment.UtilityEnvirement.XpuTcIo(1).GetMoverDetectionInfos().APM4220Expected AND
			THIS^.ipEnvironment.UtilityEnvirement.XpuTcIo(1).GetMoverDetectionInfos().APM4221Detected = THIS^.ipEnvironment.UtilityEnvirement.XpuTcIo(1).GetMoverDetectionInfos().APM4221Expected AND
			THIS^.ipEnvironment.UtilityEnvirement.XpuTcIo(1).GetMoverDetectionInfos().APM4330Detected = THIS^.ipEnvironment.UtilityEnvirement.XpuTcIo(1).GetMoverDetectionInfos().APM4330Expected AND
			THIS^.ipEnvironment.UtilityEnvirement.XpuTcIo(1).GetMoverDetectionInfos().APM4550Detected = THIS^.ipEnvironment.UtilityEnvirement.XpuTcIo(1).GetMoverDetectionInfos().APM4550Expected AND
			THIS^.ipEnvironment.UtilityEnvirement.XpuTcIo(1).GetMoverDetectionInfos().TotalDetected   = THIS^.ipEnvironment.UtilityEnvirement.XpuTcIo(1).GetMoverDetectionInfos().TotalExpected 	
		   )THEN
			nSeqEnabling := 20;
		END_IF	
			
		
		
	20: // Reset movers
		bWatchDogActive := TRUE;
		THIS^.fbMovers.ResetIterator();
		WHILE THIS^.fbMovers.HasNextObject() DO
			IF ToXpMover(THIS^.fbMovers.GetNextObject(),ipTempMover) THEN
				hr := GetMostSignificant(hr, ipTempMover.Reset());
			END_IF
		END_WHILE
		
		IF CheckOk(hr) THEN 
			nSeqEnabling := 21;
		ELSE
			nSeqEnabling := 1000 + nSeqEnabling;
		END_IF		
			
	21: // Resetting movers
		bWatchDogActive := TRUE;
		THIS^.fbMovers.ResetIterator();
		WHILE THIS^.fbMovers.HasNextObject() DO
			IF ToXpMover(THIS^.fbMovers.GetNextObject(),ipTempMover) THEN
				hr := GetMostSignificant(hr, ipTempMover.Feedback.HR);
			END_IF
		END_WHILE
		
		IF CheckOk(hr) THEN 
			nSeqEnabling := 30;
		ELSIF FAILED(hr) THEN
			nSeqEnabling := 1000 + nSeqEnabling;
		END_IF

		
		
	30: // Configure environment
		bWatchDogActive := TRUE;
		hr := ipEnvironment.Configure();
		
		IF CheckOk(hr) THEN 
			nSeqEnabling := 31;
		ELSE
			nSeqEnabling := 1000 + nSeqEnabling;
		END_IF	

	31: // Configuring environment
		bWatchDogActive := TRUE;
		hr := ipEnvironment.Feedback.HR;
		
		IF CheckOk(hr) THEN 
			nSeqEnabling := 50;
		ELSIF FAILED(hr) THEN
			nSeqEnabling := 1000 + nSeqEnabling;
		END_IF
		
		
	50: //Deside if or if not add enviroment to group
		bWatchDogActive := TRUE;
		IF XPlanarParameterlist.B_ADD_ENVIROMENT_TO_GROUP THEN
			nSeqEnabling := 51;
		ELSE
			nSeqEnabling := 70;
		END_IF
		
	51: // Add environment to group
		bWatchDogActive := TRUE;
		hr := ipEnvironment.AddToGroup(ipGroup);
		
		IF CheckOk(hr) THEN 
			nSeqEnabling := 52;
		ELSE
			nSeqEnabling := 1000 + nSeqEnabling;
		END_IF		

	52: // Adding environment to group
		bWatchDogActive := TRUE;
		hr := ipEnvironment.Feedback.HR;
		
		IF CheckOk(hr) THEN 
			nSeqEnabling := 70;
		ELSIF FAILED(hr) THEN
			nSeqEnabling := 1000 + nSeqEnabling;
		END_IF

		
	70: // Configure the tracks |
		bWatchDogActive := TRUE;
		THIS^.fbTracks.ResetIterator();
		WHILE THIS^.fbTracks.HasNextObject() DO
			IF ToXpTrack(THIS^.fbTracks.GetNextObject(),ipTempTrack) THEN
				hr := GetMostSignificant(hr, ipTempTrack.Configure());
			END_IF
		END_WHILE
		
		IF CheckOk(hr) THEN 
			nSeqEnabling := 71;
		ELSE
			nSeqEnabling := 1000 + nSeqEnabling;
		END_IF	
		
	71: // Configuring the tracks 
		bWatchDogActive := TRUE;
		THIS^.fbTracks.ResetIterator();
		WHILE THIS^.fbTracks.HasNextObject() DO
			IF ToXpTrack(THIS^.fbTracks.GetNextObject(),ipTempTrack) THEN
				hr := GetMostSignificant(hr, ipTempTrack.Configuring());
			END_IF
		END_WHILE
		
		IF CheckOk(hr) THEN 
			nSeqEnabling := 80;
		ELSIF FAILED(hr) THEN
			nSeqEnabling := 1000 + nSeqEnabling;
		END_IF	
		
		
	80: // Enable the tracks
		bWatchDogActive := TRUE;
		THIS^.fbTracks.ResetIterator();
		WHILE THIS^.fbTracks.HasNextObject() DO
			IF ToXpTrack(THIS^.fbTracks.GetNextObject(),ipTempTrack) THEN
				hr := GetMostSignificant(hr, ipTempTrack.Enable());
			END_IF
		END_WHILE
		
		IF CheckOk(hr) THEN 
			nSeqEnabling := 81;
		ELSE
			nSeqEnabling := 1000 + nSeqEnabling;
		END_IF		

	81: // Enabling the tracks
		bWatchDogActive := TRUE;
		THIS^.fbTracks.ResetIterator();
		WHILE THIS^.fbTracks.HasNextObject() DO
			IF ToXpTrack(THIS^.fbTracks.GetNextObject(),ipTempTrack) THEN
				hr := GetMostSignificant(hr, ipTempTrack.Feedback.HR);
			END_IF
		END_WHILE
		
		IF CheckOk(hr) THEN 
			nSeqEnabling := 90;
		ELSIF FAILED(hr) THEN
			nSeqEnabling := 1000 + nSeqEnabling;
		END_IF	
		
		
	90: // Add tracks to group
		bWatchDogActive := TRUE;
		THIS^.fbTracks.ResetIterator();
		WHILE THIS^.fbTracks.HasNextObject() DO
			IF ToXpTrack(THIS^.fbTracks.GetNextObject(),ipTempTrack) THEN
				hr := GetMostSignificant(hr, ipTempTrack.AddToGroup(ipGroup));
			END_IF
		END_WHILE
		
		IF CheckOk(hr) THEN 
			nSeqEnabling := 91;
		ELSE
			nSeqEnabling := 1000 + nSeqEnabling;
		END_IF	

	91: // Adding tracks to group
		bWatchDogActive := TRUE;
		THIS^.fbTracks.ResetIterator();
		WHILE THIS^.fbTracks.HasNextObject() DO
			IF ToXpTrack(THIS^.fbTracks.GetNextObject(),ipTempTrack) THEN
				hr := GetMostSignificant(hr, ipTempTrack.Feedback.HR);
			END_IF
		END_WHILE
		
		IF CheckOk(hr) THEN 
			nSeqEnabling := 100;
		ELSIF FAILED(hr) THEN
			nSeqEnabling := 1000 + nSeqEnabling;
		END_IF		
			
		
		
	100..199: // Config Station
	(* All stations are always active to the same step to ensure that all data is available in the next step.
	   The following 100 steps are defined in the station. This makes overwriting easier *)
	   
		bWatchDogActive := TRUE;
		nSupSeq := nSeqEnabling - 100;
		THIS^.fbStations.ResetIterator();
		WHILE THIS^.fbStations.HasNextObject() DO
			IF ToXpStation(THIS^.fbStations.GetNextObject(),ipTempStation) THEN
				//Call this Methode whith seq 0->99, and wait each step until S_OK is returned. Call agaiin on S_Pending
				hr := GetMostSignificant(hr, ipTempStation.Configure(nSupSeq));
			END_IF
		END_WHILE	   
	   
	   
	   	IF CheckOk(hr) AND nSupSeq >= 99 THEN
			//All steps done 
			nSeqEnabling := 210;
		ELSIF FAILED(hr) THEN
			//Error
			nSeqEnabling := 1000 + nSeqEnabling;
		ELSIF CheckOk(hr) THEN 	 
			//active step is done, continous with next
			nSeqEnabling := nSeqEnabling + 1;
		END_IF	



	210: // Enable movers
		bWatchDogActive := TRUE;
		THIS^.fbMovers.ResetIterator();
		WHILE THIS^.fbMovers.HasNextObject() DO
			IF ToXpMover(THIS^.fbMovers.GetNextObject(),ipTempMover) THEN
				hr := GetMostSignificant(hr, ipTempMover.Enable());
			END_IF
		END_WHILE
		
		IF CheckOk(hr) THEN 
			nSeqEnabling := 211;
		ELSE
			nSeqEnabling := 1000 + nSeqEnabling;
		END_IF	
		
	211: // Enabling movers
		bWatchDogActive := TRUE;
		THIS^.fbMovers.ResetIterator();
		WHILE THIS^.fbMovers.HasNextObject() DO
			IF ToXpMover(THIS^.fbMovers.GetNextObject(),ipTempMover) THEN
				hr := GetMostSignificant(hr, ipTempMover.Feedback.HR);
			END_IF
		END_WHILE
		
		IF CheckOk(hr) THEN 
			nSeqEnabling := 220;
		ELSIF FAILED(hr) THEN
			nSeqEnabling := 1000 + nSeqEnabling;
		END_IF	
		

	220: //Rotate A-Axis to zero
		bWatchDogActive := TRUE;
		THIS^.fbMovers.ResetIterator();
		WHILE THIS^.fbMovers.HasNextObject() DO
			IF ToXpMover(THIS^.fbMovers.GetNextObject(),ipTempMover) THEN
				hr := GetMostSignificant(hr, ipTempMover.MoveA(0));
			END_IF
		END_WHILE
		
		IF CheckOk(hr) THEN 
			nSeqEnabling := 221;
		ELSE
			nSeqEnabling := 1000 + nSeqEnabling;
		END_IF	
		
	221: //Rotating A-Axis to Zero	
		bWatchDogActive := TRUE;		
		THIS^.fbMovers.ResetIterator();
		WHILE THIS^.fbMovers.HasNextObject() DO
			IF ToXpMover(THIS^.fbMovers.GetNextObject(),ipTempMover) THEN
				hr := GetMostSignificant(hr, ipTempMover.Feedback.HR);
			END_IF
		END_WHILE
		
		IF CheckOk(hr) THEN 
			nSeqEnabling := 222;
		ELSIF FAILED(hr) THEN
			nSeqEnabling := 1000 + nSeqEnabling;
		END_IF	
		
	222: //Rotate B-Axis to zero
		bWatchDogActive := TRUE;
		THIS^.fbMovers.ResetIterator();
		WHILE THIS^.fbMovers.HasNextObject() DO
			IF ToXpMover(THIS^.fbMovers.GetNextObject(),ipTempMover) THEN
				hr := GetMostSignificant(hr, ipTempMover.MoveB(0));
			END_IF
		END_WHILE
		
		IF CheckOk(hr) THEN 
			nSeqEnabling := 223;
		ELSE
			nSeqEnabling := 1000 + nSeqEnabling;
		END_IF	
		
	223: //Rotating B-Axis to zero
		bWatchDogActive := TRUE;			
		THIS^.fbMovers.ResetIterator();
		WHILE THIS^.fbMovers.HasNextObject() DO
			IF ToXpMover(THIS^.fbMovers.GetNextObject(),ipTempMover) THEN
				hr := GetMostSignificant(hr, ipTempMover.Feedback.HR);
			END_IF
		END_WHILE
		
		IF CheckOk(hr) THEN 
			nSeqEnabling := 230;
		ELSIF FAILED(hr) THEN
			nSeqEnabling := 1000 + nSeqEnabling;
		END_IF		
		
				
		
	230: //Rotate C-Axis to "Zero" (to the next 90 degree pitch)
		bWatchDogActive := TRUE;
		THIS^.fbMovers.ResetIterator();
		WHILE THIS^.fbMovers.HasNextObject() DO
			IF ToXpMover(THIS^.fbMovers.GetNextObject(),ipTempMover) THEN
				// Decide which 90 degree pitch is closer to the current position. If the remainder is greater than 45 degrees, then round up to the next 90 degree division.
				lrCRotationShortestPos := LREAL_TO_DINT(ipTempMover.PlanarMover.MCTOPLC.SET.SetPos.C / 90.0) * 90.0;
				hr := GetMostSignificant(hr, ipTempMover.MoveC(	fPosition		:= lrCRotationShortestPos, 
																additionalTurns := 0,
																direction		:= Tc3_Mc3Definitions.MC_DIRECTION.mcDirectionShortestWay));
			END_IF
		END_WHILE
		
		IF CheckOk(hr) THEN 
			nSeqEnabling := 231;
		ELSE
			nSeqEnabling := 1000 + nSeqEnabling;
		END_IF	
		
	231: //Rotating C-Axis to Zero		
		bWatchDogActive := TRUE;	
		THIS^.fbMovers.ResetIterator();
		WHILE THIS^.fbMovers.HasNextObject() DO
			IF ToXpMover(THIS^.fbMovers.GetNextObject(),ipTempMover) THEN
				hr := GetMostSignificant(hr, ipTempMover.Feedback.HR);
			END_IF
		END_WHILE
		
		IF CheckOk(hr) THEN 
			nSeqEnabling := 240;
		ELSIF FAILED(hr) THEN
			nSeqEnabling := 1000 + nSeqEnabling;
		END_IF	
			
		
		
	240: // Add movers to group
		bWatchDogActive := TRUE;
		THIS^.fbMovers.ResetIterator();
		WHILE THIS^.fbMovers.HasNextObject() DO
			IF ToXpMover(THIS^.fbMovers.GetNextObject(),ipTempMover) THEN
				hr := GetMostSignificant(hr, ipTempMover.AddToGroup(THIS^.ipGroup));
			END_IF
		END_WHILE
		
		IF CheckOk(hr) THEN 
			nSeqEnabling := 241;
		ELSE
			nSeqEnabling := 1000 + nSeqEnabling;
		END_IF	
	
	241: // Adding mover to group
		bWatchDogActive := TRUE;
		THIS^.fbMovers.ResetIterator();
		WHILE THIS^.fbMovers.HasNextObject() DO
			IF ToXpMover(THIS^.fbMovers.GetNextObject(),ipTempMover) THEN
				hr := GetMostSignificant(hr, ipTempMover.Feedback.HR);
			END_IF
		END_WHILE
		
		IF CheckOk(hr) THEN 
			nSeqEnabling := 300;
		ELSIF FAILED(hr) THEN
			nSeqEnabling := 1000 + nSeqEnabling;
		END_IF		
	
		
		
	300: // Enable group
		bWatchDogActive := TRUE;
		hr := ipGroup.Enable();
		
		IF CheckOk(hr) THEN 
			nSeqEnabling := 310;
		ELSE
			nSeqEnabling := 1000 + nSeqEnabling;
		END_IF	
		
	310: // Enabling group
		bWatchDogActive := TRUE;
		hr := ipGroup.Feedback.HR;
		
		IF CheckOk(hr) THEN 
			nSeqEnabling := 400;
		ELSIF FAILED(hr) THEN
			nSeqEnabling := 1000 + nSeqEnabling;
		END_IF	

		
		
		
	400: (*	Restart of the sequenze "JoiningTrack". Default strategy is that each mover joins the closest track
			Outsourced to a method for easier overwriting *)
		THIS^.nSeqJoiningTrack := 0;	
		nSeqEnabling := 401;	

	401: (*	Default strategy is that each mover joins the closest track
			Outsourced to a method for easier overwriting *)
		hr := THIS^.JoiningTrack();

		IF CheckOk(hr) THEN 
			nSeqEnabling := 500;
		ELSIF FAILED(hr) THEN
			nSeqEnabling := 1000 + nSeqEnabling;
		END_IF	
		
	

	
	500: (*	Restart of the sequenze "JoiningStation" to distribute the movers to the available stations.
			Outsourced to a method for easier overwriting *)
		THIS^.nSeqJoiningStation := 0;	
		nSeqEnabling := 501;	
	
	501: (*	Distribute the movers to the available stations.
		 	Outsourced to a method for easier overwriting *)
		hr := THIS^.JoiningStation();

		IF CheckOk(hr) THEN 
			nSeqEnabling := SEQ_DONE;
		ELSIF FAILED(hr) THEN
			nSeqEnabling := 1000 + nSeqEnabling;
		END_IF	


		
		
	SEQ_DONE: // Done
		Enabling := S_OK;

		
	1000..1999://Error
		hr := GetMostSignificant(hrLastCycle, E_FAIL);
		//Only rais if timeout is not active
		IF NOT fbErrorEnabling.bRaised AND NOT fbTimeOutEnabling.bRaised THEN 
			fbErrorEnabling.CreateEx(stEventEntry:=TC_EVENTS.CHALET_XPlanar_Events.ErrorEnabling, ipSourceInfo := THIS^.fbSourceInfo, bWithConfirmation := FALSE);
			fbErrorEnabling.ipArguments.AddUInt(nSeqEnabling-1000);
			fbErrorEnabling.Raise(0);
		END_IF
END_CASE


//Timeout after to long stay in one of the following seq.
fbTimeOutSeq.IN := (nlastState = nSeqEnabling) AND bWatchDogActive;
fbTimeOutSeq.PT := T#5S;
fbTimeOutSeq();
nlastState := nSeqEnabling;

IF fbTimeOutSeq.Q THEN
	IF NOT fbTimeOutEnabling.bRaised THEN 
		fbTimeOutEnabling.CreateEx(stEventEntry:=TC_EVENTS.CHALET_XPlanar_Events.TimeOutEnabling, ipSourceInfo := THIS^.fbSourceInfo, bWithConfirmation := FALSE);
		fbTimeOutEnabling.ipArguments.AddUInt(nSeqEnabling);
		fbTimeOutEnabling.Raise(0);
	END_IF
	//next seq is error
	nSeqEnabling := 1000 + nSeqEnabling;
END_IF

//Clear Tc3-Eventlogger alarm 
IF nSeqEnabling <= SEQ_DONE THEN
	fbTimeOutEnabling.Clear(0,0);
	fbErrorEnabling.Clear(0,0);
END_IF


//store last information
hrLastCycle := hr;

// Propagate error
IF FAILED(hr) THEN
	Enabling := hr;
END_IF
END_METHOD

